KUKA KRL program: EPS_2_25716_MHDR04_A_20250926070356.src

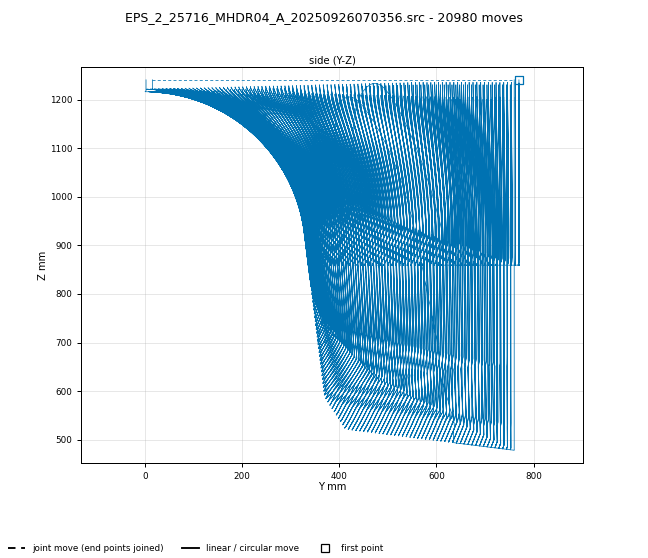
[picture p0: tool path of EPS_2_25716_MHDR04_A_20250926070356.src, 20980 of 20982 moves have a stored position in this frame; points joined in program order, loops and branches not executed]
&ACCESS RVP
&REL 4
&COMMENT QRS 19112012
&PARAM EDITMASK = *
DEF PART()
EXT BAS (BAS_COMMAND :IN,REAL :IN )
INT I
BAS (#INITMOV,0 )

;KUKA QRS Post kuka4.cps  Date:22-06-2017 !

File_ID=2853

QRS_PRE_INIT()

;Init var - Until changes are made in qrs_pre_init
Outlet_Square_prg=0
Inlet_1_Square_prg=0
Inlet_2_Square_prg=0
Inlet_3_Square_prg=0
Inlet_4_Square_prg=0
Inlet_5_Square_prg=0

Outlet_1={X 0.000, Y 562.000, Z 887.500, B 0.000, E1 0.000 }
Inlet_1={X 0.000, Y 612.000, Z 934.000, B 0.000, E1 180.000 }
Outlet_1_type=686
Inlet_1_type=533
;QRS#1=Sidecore dimensions
;QRS#2=675-27" Concrete
;QRS#3=525-21" Concrete
;QRS#4=
;QRS#5=
;QRS#6=
;QRS#7=
;QRS#8=
;QRS#9=S306-38L
;QRS#10=S306-32
;QRS#11=
;QRS#12=
;QRS#13=
;QRS#14=
;QRS#15=
;QRS#16=1524x152x1676 5,5'
;QRS#17=EPS Height
;QRS#18=1230,5
;QRS#19=*
;QRS#20= UPDATED VERSION 22-06-2017
;QRS#21=*
Outlet_Square=0550
Inlet_1_Square=0350
Inlet_2_Square=0
Inlet_3_Square=0
Inlet_4_Square=0
Inlet_5_Square=0
Mill_Square=1
Outlet_Square_Prg=265
Inlet_1_Square_prg=263

QRS_INIT()

$ADVANCE=5

; T1
PTP {E1 171.906,E2 171.906}
PTP {X 0,Y 769.671,A -85,B 0,C 180,E1 171.906,E2 171.906,E3 0,E4 0,E5 0,E6 0}
QRS_SPEED_INIT()
LIN {X 0,Y 769.671,Z 1240.5,A -85,B 0,C 180,E1 171.906,E2 171.906,E3 0,E4 0,E5 0,E6 0} C_VEL
LIN {X 0,Y 769.671,Z 861.31,A -85,B 0,C 180,E1 171.906,E2 171.906} C_VEL
LIN {X 0,Y 769.682,Z 859.31,A -85,B 0,C 180,E1 172.055,E2 172.055} C_VEL
LIN {X 0,Y 770.051,Z 859.31,A -85,B 0,C 180,E1 173.477,E2 173.477} C_VEL
LIN {X 0,Y 770.066,Z 859.31,A -85,B 0,C 180,E1 177.209,E2 177.209} C_VEL
LIN {X 0,Y 770.077,Z 859.31,A -85,B 0,C 180,E1 180.93,E2 180.93} C_VEL
LIN {X 0,Y 770.044,Z 859.31,A -85,B 0,C 180,E1 184.654,E2 184.654} C_VEL
LIN {X 0,Y 770.001,Z 859.31,A -85,B 0,C 180,E1 188.399,E2 188.399} C_VEL
LIN {X 0,Y 769.978,Z 859.31,A -85,B 0,C 180,E1 192.181,E2 192.181} C_VEL
LIN {X 0,Y 769.977,Z 859.31,A -85,B 0,C 180,E1 196.017,E2 196.017} C_VEL
LIN {X 0,Y 769.85,Z 859.31,A -85,B 0,C 180,E1 196.72,E2 196.72} C_VEL
LIN {X 0,Y 769.988,Z 859.31,A -85,B 0,C 180,E1 199.928,E2 199.928} C_VEL
LIN {X 0,Y 769.595,Z 859.31,A -85,B 0,C 180,E1 202.247,E2 202.247} C_VEL
LIN {X 0,Y 769.967,Z 859.31,A -85,B 0,C 180,E1 203.939,E2 203.939} C_VEL
LIN {X 0,Y 769.591,Z 859.31,A -85,B 0,C 180,E1 206.736,E2 206.736} C_VEL
LIN {X 0,Y 769.937,Z 859.31,A -85,B 0,C 180,E1 208.08,E2 208.08} C_VEL
LIN {X 0,Y 769.495,Z 859.31,A -85,B 0,C 180,E1 210.602,E2 210.602} C_VEL
LIN {X 0,Y 769.877,Z 859.31,A -85,B 0,C 180,E1 212.39,E2 212.39} C_VEL
LIN {X 0,Y 769.44,Z 859.31,A -85,B 0,C 180,E1 214.643,E2 214.643} C_VEL
LIN {X 0,Y 770.006,Z 859.31,A -85,B 0,C 180,E1 217.323,E2 217.323} C_VEL
LIN {X 0,Y 769.695,Z 859.31,A -85,B 0,C 180,E1 221.735,E2 221.735} C_VEL
LIN {X 0,Y 769.74,Z 859.31,A -85,B 0,C 180,E1 223.066,E2 223.066} C_VEL
LIN {X 0,Y 769.705,Z 859.31,A -85,B 0,C 180,E1 226.939,E2 226.939} C_VEL
LIN {X 0,Y 769.666,Z 859.31,A -85,B 0,C 180,E1 228.264,E2 228.264} C_VEL
LIN {X 0,Y 770.07,Z 859.31,A -85,B 0,C 180,E1 232.674,E2 232.674} C_VEL
LIN {X 0,Y 769.756,Z 859.31,A -85,B 0,C 180,E1 235.893,E2 235.893} C_VEL
LIN {X 0,Y 769.798,Z 859.31,A -85,B 0,C 180,E1 237.608,E2 237.608} C_VEL
LIN {X 0,Y 770.017,Z 859.31,A -85,B 0,C 180,E1 240.258,E2 240.258} C_VEL
LIN {X 0,Y 769.761,Z 859.31,A -85,B 0,C 180,E1 240.478,E2 240.478} C_VEL
LIN {X 0,Y 767.984,Z 859.31,A -85,B 0,C 180,E1 240.653,E2 240.653} C_VEL
LIN {X 0,Y 768.026,Z 859.947,A -85,B 0,C 180,E1 240.678,E2 240.678} C_VEL
LIN {X 0,Y 769.267,Z 864.427,A -85,B 0,C 180,E1 240.777,E2 240.777} C_VEL
LIN {X 0,Y 769.568,Z 866.732,A -85,B 0,C 180,E1 240.814,E2 240.814} C_VEL
LIN {X 0,Y 769.716,Z 904.713,A -85,B 0,C 180,E1 241.217,E2 241.217} C_VEL
LIN {X 0,Y 769.839,Z 924.965,A -85,B 0,C 180,E1 241.466,E2 241.466} C_VEL
LIN {X 0,Y 769.627,Z 943.026,A -85,B 0,C 180,E1 241.759,E2 241.759} C_VEL
LIN {X 0,Y 769.796,Z 960.577,A -85,B 0,C 180,E1 242.132,E2 242.132} C_VEL
LIN {X 0,Y 769.69,Z 975.698,A -85,B 0,C 180,E1 242.501,E2 242.501} C_VEL
LIN {X 0,Y 769.872,Z 993.181,A -85,B 0,C 180,E1 243.017,E2 243.017} C_VEL
LIN {X 0,Y 769.856,Z 1009.123,A -85,B 0,C 180,E1 243.548,E2 243.548} C_VEL
LIN {X 0,Y 769.815,Z 1019.932,A -85,B 0,C 180,E1 243.947,E2 243.947} C_VEL
LIN {X 0,Y 769.91,Z 1034.617,A -85,B 0,C 180,E1 244.55,E2 244.55} C_VEL
LIN {X 0,Y 769.91,Z 1042.438,A -85,B 0,C 180,E1 244.896,E2 244.896} C_VEL
LIN {X 0,Y 769.862,Z 1054.848,A -85,B 0,C 180,E1 245.478,E2 245.478} C_VEL
LIN {X 0,Y 769.906,Z 1068.593,A -85,B 0,C 180,E1 246.187,E2 246.187} C_VEL
LIN {X 0,Y 769.93,Z 1082.086,A -85,B 0,C 180,E1 246.948,E2 246.948} C_VEL
LIN {X 0,Y 769.915,Z 1094.982,A -85,B 0,C 180,E1 247.739,E2 247.739} C_VEL
LIN {X 0,Y 769.892,Z 1107.85,A -85,B 0,C 180,E1 248.6,E2 248.6} C_VEL
LIN {X 0,Y 769.939,Z 1119.711,A -85,B 0,C 180,E1 249.464,E2 249.464} C_VEL
LIN {X 0,Y 769.935,Z 1130.574,A -85,B 0,C 180,E1 250.319,E2 250.319} C_VEL
LIN {X 0,Y 769.888,Z 1142.058,A -85,B 0,C 180,E1 251.302,E2 251.302} C_VEL
LIN {X 0,Y 769.98,Z 1153.138,A -85,B 0,C 180,E1 252.343,E2 252.343} C_VEL
LIN {X 0,Y 769.834,Z 1162.511,A -85,B 0,C 180,E1 253.29,E2 253.29} C_VEL
LIN {X 0,Y 769.848,Z 1172.264,A -85,B 0,C 180,E1 254.376,E2 254.376} C_VEL
LIN {X 0,Y 769.964,Z 1181.174,A -85,B 0,C 180,E1 255.469,E2 255.469} C_VEL
LIN {X 0,Y 769.771,Z 1189.787,A -85,B 0,C 180,E1 256.624,E2 256.624} C_VEL
LIN {X 0,Y 769.791,Z 1196.239,A -85,B 0,C 180,E1 257.579,E2 257.579} C_VEL
LIN {X 0,Y 769.97,Z 1203.41,A -85,B 0,C 180,E1 258.769,E2 258.769} C_VEL
LIN {X 0,Y 769.805,Z 1209.797,A -85,B 0,C 180,E1 259.95,E2 259.95} C_VEL
LIN {X 0,Y 769.942,Z 1216.32,A -85,B 0,C 180,E1 261.365,E2 261.365} C_VEL
LIN {X 0,Y 769.923,Z 1219.537,A -85,B 0,C 180,E1 262.168,E2 262.168} C_VEL
LIN {X 0,Y 769.786,Z 1222.09,A -85,B 0,C 180,E1 262.857,E2 262.857} C_VEL
LIN {X 0,Y 769.781,Z 1225.359,A -85,B 0,C 180,E1 263.849,E2 263.849} C_VEL
LIN {X 0,Y 769.875,Z 1227.368,A -85,B 0,C 180,E1 264.598,E2 264.598} C_VEL
LIN {X 0,Y 769.915,Z 1229.173,A -85,B 0,C 180,E1 265.345,E2 265.345} C_VEL
LIN {X 0,Y 769.759,Z 1230.789,A -85,B 0,C 180,E1 266.09,E2 266.09} C_VEL
LIN {X 0,Y 769.725,Z 1232.561,A -85,B 0,C 180,E1 267.208,E2 267.208} C_VEL
LIN {X 0,Y 769.922,Z 1233.68,A -85,B 0,C 180,E1 268.326,E2 268.326} C_VEL
LIN {X 0,Y 769.882,Z 1234.171,A -85,B 0,C 180,E1 269.07,E2 269.07} C_VEL
LIN {X 0,Y 769.752,Z 1234.206,A -85,B 0,C 180,E1 270.93,E2 270.93} C_VEL
LIN {X 0,Y 769.983,Z 1233.333,A -85,B 0,C 180,E1 272.046,E2 272.046} C_VEL
LIN {X 0,Y 769.853,Z 1232.527,A -85,B 0,C 180,E1 272.791,E2 272.791} C_VEL
LIN {X 0,Y 769.748,Z 1230.792,A -85,B 0,C 180,E1 273.91,E2 273.91} C_VEL
LIN {X 0,Y 769.834,Z 1229.195,A -85,B 0,C 180,E1 274.656,E2 274.656} C_VEL
LIN {X 0,Y 769.978,Z 1227.341,A -85,B 0,C 180,E1 275.401,E2 275.401} C_VEL
LIN {X 0,Y 769.82,Z 1225.349,A -85,B 0,C 180,E1 276.15,E2 276.15} C_VEL
LIN {X 0,Y 769.746,Z 1221.269,A -85,B 0,C 180,E1 277.393,E2 277.393} C_VEL
LIN {X 0,Y 769.943,Z 1215.307,A -85,B 0,C 180,E1 278.87,E2 278.87} C_VEL
LIN {X 0,Y 769.789,Z 1209.8,A -85,B 0,C 180,E1 280.05,E2 280.05} C_VEL
LIN {X 0,Y 769.876,Z 1203.431,A -85,B 0,C 180,E1 281.232,E2 281.232} C_VEL
LIN {X 0,Y 769.918,Z 1197.677,A -85,B 0,C 180,E1 282.181,E2 282.181} C_VEL
LIN {X 0,Y 769.805,Z 1193.003,A -85,B 0,C 180,E1 282.898,E2 282.898} C_VEL
LIN {X 0,Y 769.803,Z 1188.107,A -85,B 0,C 180,E1 283.614,E2 283.614} C_VEL
LIN {X 0,Y 769.984,Z 1178.906,A -85,B 0,C 180,E1 284.816,E2 284.816} C_VEL
LIN {X 0,Y 769.839,Z 1170.607,A -85,B 0,C 180,E1 285.819,E2 285.819} C_VEL
LIN {X 0,Y 769.821,Z 1160.767,A -85,B 0,C 180,E1 286.894,E2 286.894} C_VEL
LIN {X 0,Y 769.967,Z 1150.001,A -85,B 0,C 180,E1 287.961,E2 287.961} C_VEL
LIN {X 0,Y 769.878,Z 1139.267,A -85,B 0,C 180,E1 288.944,E2 288.944} C_VEL
LIN {X 0,Y 769.906,Z 1129.048,A -85,B 0,C 180,E1 289.806,E2 289.806} C_VEL
LIN {X 0,Y 769.942,Z 1116.517,A -85,B 0,C 180,E1 290.773,E2 290.773} C_VEL
LIN {X 0,Y 769.9,Z 1105.284,A -85,B 0,C 180,E1 291.577,E2 291.577} C_VEL
LIN {X 0,Y 769.914,Z 1092.612,A -85,B 0,C 180,E1 292.411,E2 292.411} C_VEL
LIN {X 0,Y 769.921,Z 1078.814,A -85,B 0,C 180,E1 293.242,E2 293.242} C_VEL
LIN {X 0,Y 769.909,Z 1064.631,A -85,B 0,C 180,E1 294.023,E2 294.023} C_VEL
LIN {X 0,Y 769.846,Z 1051.463,A -85,B 0,C 180,E1 294.69,E2 294.69} C_VEL
LIN {X 0,Y 769.909,Z 1036.961,A -85,B 0,C 180,E1 295.353,E2 295.353} C_VEL
LIN {X 0,Y 769.869,Z 1020.065,A -85,B 0,C 180,E1 296.046,E2 296.046} C_VEL
LIN {X 0,Y 769.811,Z 1007.364,A -85,B 0,C 180,E1 296.519,E2 296.519} C_VEL
LIN {X 0,Y 769.897,Z 989.325,A -85,B 0,C 180,E1 297.102,E2 297.102} C_VEL
LIN {X 0,Y 769.783,Z 972.607,A -85,B 0,C 180,E1 297.575,E2 297.575} C_VEL
LIN {X 0,Y 769.703,Z 963.365,A -85,B 0,C 180,E1 297.804,E2 297.804} C_VEL
LIN {X 0,Y 769.829,Z 954.273,A -85,B 0,C 180,E1 298.005,E2 298.005} C_VEL
LIN {X 0,Y 769.853,Z 939.702,A -85,B 0,C 180,E1 298.293,E2 298.293} C_VEL
LIN {X 0,Y 769.612,Z 922.786,A -85,B 0,C 180,E1 298.571,E2 298.571} C_VEL
LIN {X 0,Y 769.691,Z 903.386,A -85,B 0,C 180,E1 298.798,E2 298.798} C_VEL
LIN {X 0,Y 769.594,Z 868.345,A -85,B 0,C 180,E1 299.168,E2 299.168} C_VEL
LIN {X 0,Y 769.47,Z 865.258,A -85,B 0,C 180,E1 299.206,E2 299.206} C_VEL
LIN {X 0,Y 768.381,Z 860.967,A -85,B 0,C 180,E1 299.296,E2 299.296} C_VEL
LIN {X 0,Y 767.894,Z 859.31,A -85,B 0,C 180,E1 299.344,E2 299.344} C_VEL
LIN {X 0,Y 768.202,Z 859.31,A -85,B 0,C 180,E1 299.358,E2 299.358} C_VEL
LIN {X 0,Y 769.579,Z 859.31,A -85,B 0,C 180,E1 299.487,E2 299.487} C_VEL
LIN {X 0,Y 770.036,Z 859.31,A -85,B 0,C 180,E1 299.696,E2 299.696} C_VEL
LIN {X 0,Y 769.962,Z 859.31,A -85,B 0,C 180,E1 302.384,E2 302.384} C_VEL
LIN {X 0,Y 769.489,Z 859.31,A -85,B 0,C 180,E1 304.639,E2 304.639} C_VEL
LIN {X 0,Y 770.073,Z 859.31,A -85,B 0,C 180,E1 307.326,E2 307.326} C_VEL
LIN {X 0,Y 769.766,Z 859.31,A -85,B 0,C 180,E1 311.729,E2 311.729} C_VEL
LIN {X 0,Y 769.826,Z 859.31,A -85,B 0,C 180,E1 313.071,E2 313.071} C_VEL
LIN {X 0,Y 769.84,Z 859.31,A -85,B 0,C 180,E1 314.267,E2 314.267} C_VEL
LIN {X 0,Y 769.763,Z 859.31,A -85,B 0,C 180,E1 315.725,E2 315.725} C_VEL
LIN {X 0,Y 769.763,Z 859.31,A -85,B 0,C 180,E1 319.731,E2 319.731} C_VEL
LIN {X 0,Y 769.807,Z 859.31,A -85,B 0,C 180,E1 320.719,E2 320.719} C_VEL
LIN {X 0,Y 769.409,Z 859.31,A -85,B 0,C 180,E1 323.061,E2 323.061} C_VEL
LIN {X 0,Y 769.837,Z 859.31,A -85,B 0,C 180,E1 325.377,E2 325.377} C_VEL
LIN {X 0,Y 770.001,Z 859.31,A -85,B 0,C 180,E1 329.334,E2 329.334} C_VEL
LIN {X 0,Y 769.842,Z 859.31,A -85,B 0,C 180,E1 333.227,E2 333.227} C_VEL
LIN {X 0,Y 769.935,Z 859.31,A -85,B 0,C 180,E1 334.008,E2 334.008} C_VEL
LIN {X 0,Y 769.999,Z 859.31,A -85,B 0,C 180,E1 337.68,E2 337.68} C_VEL
LIN {X 0,Y 769.97,Z 859.31,A -85,B 0,C 180,E1 338.08,E2 338.08} C_VEL
LIN {X 0,Y 769.98,Z 859.31,A -85,B 0,C 180,E1 342.039,E2 342.039} C_VEL
LIN {X 0,Y 769.696,Z 859.31,A -85,B 0,C 180,E1 343.977,E2 343.977} C_VEL
LIN {X 0,Y 769.78,Z 859.31,A -85,B 0,C 180,E1 345.906,E2 345.906} C_VEL
LIN {X 0,Y 769.98,Z 859.31,A -85,B 0,C 180,E1 349.716,E2 349.716} C_VEL
LIN {X 0,Y 770.006,Z 859.31,A -85,B 0,C 180,E1 353.477,E2 353.477} C_VEL
LIN {X 0,Y 770.059,Z 859.31,A -85,B 0,C 180,E1 357.209,E2 357.209} C_VEL
LIN {X 0,Y 770.073,Z 859.31,A -85,B 0,C 180,E1 360.93,E2 360.93} C_VEL
LIN {X 0,Y 770.057,Z 859.31,A -85,B 0,C 180,E1 364.654,E2 364.654} C_VEL
LIN {X 0,Y 770.018,Z 859.31,A -85,B 0,C 180,E1 368.399,E2 368.399} C_VEL
LIN {X 0,Y 769.982,Z 859.31,A -85,B 0,C 180,E1 372.181,E2 372.181} C_VEL
LIN {X 0,Y 769.963,Z 859.31,A -85,B 0,C 180,E1 376.017,E2 376.017} C_VEL
LIN {X 0,Y 769.829,Z 859.31,A -85,B 0,C 180,E1 376.715,E2 376.715} C_VEL
LIN {X 0,Y 769.937,Z 859.31,A -85,B 0,C 180,E1 379.929,E2 379.929} C_VEL
LIN {X 0,Y 769.562,Z 859.31,A -85,B 0,C 180,E1 382.241,E2 382.241} C_VEL
LIN {X 0,Y 769.917,Z 859.31,A -85,B 0,C 180,E1 383.941,E2 383.941} C_VEL
LIN {X 0,Y 769.542,Z 859.31,A -85,B 0,C 180,E1 386.729,E2 386.729} C_VEL
LIN {X 0,Y 769.888,Z 859.31,A -85,B 0,C 180,E1 388.082,E2 388.082} C_VEL
LIN {X 0,Y 769.488,Z 859.31,A -85,B 0,C 180,E1 390.601,E2 390.601} C_VEL
LIN {X 0,Y 769.865,Z 859.31,A -85,B 0,C 180,E1 392.39,E2 392.39} C_VEL
LIN {X 0,Y 769.445,Z 859.31,A -85,B 0,C 180,E1 394.643,E2 394.643} C_VEL
LIN {X 0,Y 770.04,Z 859.31,A -85,B 0,C 180,E1 397.326,E2 397.326} C_VEL
LIN {X 0,Y 769.705,Z 859.31,A -85,B 0,C 180,E1 401.735,E2 401.735} C_VEL
LIN {X 0,Y 769.752,Z 859.31,A -85,B 0,C 180,E1 403.067,E2 403.067} C_VEL
LIN {X 0,Y 769.737,Z 859.31,A -85,B 0,C 180,E1 406.937,E2 406.937} C_VEL
LIN {X 0,Y 769.692,Z 859.31,A -85,B 0,C 180,E1 408.266,E2 408.266} C_VEL
LIN {X 0,Y 770.062,Z 859.31,A -85,B 0,C 180,E1 412.675,E2 412.675} C_VEL
LIN {X 0,Y 769.748,Z 859.31,A -85,B 0,C 180,E1 415.894,E2 415.894} C_VEL
LIN {X 0,Y 769.672,Z 859.31,A -85,B 0,C 180,E1 417.602,E2 417.602} C_VEL
LIN {X 0,Y 769.433,Z 859.31,A -85,B 0,C 180,E1 419.769,E2 419.769} C_VEL
LIN {X 0,Y 769.91,Z 859.31,A -85,B 0,C 180,E1 421.92,E2 421.92} C_VEL
LIN {X 0,Y 770.081,Z 859.31,A -85,B 0,C 180,E1 426.297,E2 426.297} C_VEL
LIN {X 0,Y 769.403,Z 859.31,A -85,B 0,C 180,E1 426.506,E2 426.506} C_VEL
LIN {X 0,Y 768.639,Z 859.31,A -85,B 0,C 180,E1 426.577,E2 426.577} C_VEL
LIN {X 0,Y 769.411,Z 862.963,A -85,B 0,C 180,E1 426.652,E2 426.652} C_VEL
LIN {X 0,Y 769.765,Z 870.896,A -85,B 0,C 180,E1 426.742,E2 426.742} C_VEL
LIN {X 0,Y 769.853,Z 946.408,A -85,B 0,C 180,E1 427.495,E2 427.495} C_VEL
LIN {X 0,Y 769.952,Z 960.871,A -85,B 0,C 180,E1 427.677,E2 427.677} C_VEL
LIN {X 0,Y 769.864,Z 974.295,A -85,B 0,C 180,E1 427.892,E2 427.892} C_VEL
LIN {X 0,Y 769.934,Z 984.387,A -85,B 0,C 180,E1 428.089,E2 428.089} C_VEL
LIN {X 0,Y 769.985,Z 999.962,A -85,B 0,C 180,E1 428.458,E2 428.458} C_VEL
LIN {X 0,Y 769.905,Z 1013.381,A -85,B 0,C 180,E1 428.83,E2 428.83} C_VEL
LIN {X 0,Y 769.957,Z 1025.148,A -85,B 0,C 180,E1 429.206,E2 429.206} C_VEL
LIN {X 0,Y 769.979,Z 1038.217,A -85,B 0,C 180,E1 429.68,E2 429.68} C_VEL
LIN {X 0,Y 769.926,Z 1049.488,A -85,B 0,C 180,E1 430.133,E2 430.133} C_VEL
LIN {X 0,Y 769.981,Z 1061.815,A -85,B 0,C 180,E1 430.69,E2 430.69} C_VEL
LIN {X 0,Y 769.982,Z 1072.942,A -85,B 0,C 180,E1 431.243,E2 431.243} C_VEL
LIN {X 0,Y 769.967,Z 1084.12,A -85,B 0,C 180,E1 431.855,E2 431.855} C_VEL
LIN {X 0,Y 769.957,Z 1094.576,A -85,B 0,C 180,E1 432.483,E2 432.483} C_VEL
LIN {X 0,Y 769.955,Z 1104.699,A -85,B 0,C 180,E1 433.149,E2 433.149} C_VEL
LIN {X 0,Y 769.998,Z 1113.725,A -85,B 0,C 180,E1 433.794,E2 433.794} C_VEL
LIN {X 0,Y 769.959,Z 1123.75,A -85,B 0,C 180,E1 434.577,E2 434.577} C_VEL
LIN {X 0,Y 769.898,Z 1131.942,A -85,B 0,C 180,E1 435.272,E2 435.272} C_VEL
LIN {X 0,Y 769.96,Z 1140.118,A -85,B 0,C 180,E1 436.029,E2 436.029} C_VEL
LIN {X 0,Y 769.949,Z 1148.387,A -85,B 0,C 180,E1 436.866,E2 436.866} C_VEL
LIN {X 0,Y 769.87,Z 1155.915,A -85,B 0,C 180,E1 437.699,E2 437.699} C_VEL
LIN {X 0,Y 769.914,Z 1162.733,A -85,B 0,C 180,E1 438.531,E2 438.531} C_VEL
LIN {X 0,Y 769.978,Z 1168.094,A -85,B 0,C 180,E1 439.243,E2 439.243} C_VEL
LIN {X 0,Y 769.844,Z 1174.555,A -85,B 0,C 180,E1 440.186,E2 440.186} C_VEL
LIN {X 0,Y 769.866,Z 1180.255,A -85,B 0,C 180,E1 441.129,E2 441.129} C_VEL
LIN {X 0,Y 769.951,Z 1185.836,A -85,B 0,C 180,E1 442.192,E2 442.192} C_VEL
LIN {X 0,Y 769.81,Z 1190.358,A -85,B 0,C 180,E1 443.172,E2 443.172} C_VEL
LIN {X 0,Y 769.845,Z 1194.421,A -85,B 0,C 180,E1 444.224,E2 444.224} C_VEL
LIN {X 0,Y 769.974,Z 1196.895,A -85,B 0,C 180,E1 444.972,E2 444.972} C_VEL
LIN {X 0,Y 769.82,Z 1199.939,A -85,B 0,C 180,E1 446.091,E2 446.091} C_VEL
LIN {X 0,Y 769.843,Z 1202.142,A -85,B 0,C 180,E1 447.209,E2 447.209} C_VEL
LIN {X 0,Y 769.986,Z 1203.212,A -85,B 0,C 180,E1 447.954,E2 447.954} C_VEL
LIN {X 0,Y 769.799,Z 1204.215,A -85,B 0,C 180,E1 449.07,E2 449.07} C_VEL
LIN {X 0,Y 769.84,Z 1204.172,A -85,B 0,C 180,E1 450.93,E2 450.93} C_VEL
LIN {X 0,Y 769.988,Z 1203.478,A -85,B 0,C 180,E1 451.674,E2 451.674} C_VEL
LIN {X 0,Y 769.807,Z 1202.02,A -85,B 0,C 180,E1 452.791,E2 452.791} C_VEL
LIN {X 0,Y 769.853,Z 1199.737,A -85,B 0,C 180,E1 453.909,E2 453.909} C_VEL
LIN {X 0,Y 769.949,Z 1196.599,A -85,B 0,C 180,E1 455.028,E2 455.028} C_VEL
LIN {X 0,Y 769.846,Z 1194.12,A -85,B 0,C 180,E1 455.776,E2 455.776} C_VEL
LIN {X 0,Y 769.885,Z 1190.021,A -85,B 0,C 180,E1 456.818,E2 456.818} C_VEL
LIN {X 0,Y 769.948,Z 1185.617,A -85,B 0,C 180,E1 457.765,E2 457.765} C_VEL
LIN {X 0,Y 769.837,Z 1179.731,A -85,B 0,C 180,E1 458.871,E2 458.871} C_VEL
LIN {X 0,Y 769.928,Z 1173.935,A -85,B 0,C 180,E1 459.812,E2 459.812} C_VEL
LIN {X 0,Y 769.961,Z 1167.417,A -85,B 0,C 180,E1 460.757,E2 460.757} C_VEL
LIN {X 0,Y 769.874,Z 1160.128,A -85,B 0,C 180,E1 461.707,E2 461.707} C_VEL
LIN {X 0,Y 769.934,Z 1153.042,A -85,B 0,C 180,E1 462.538,E2 462.538} C_VEL
LIN {X 0,Y 769.957,Z 1145.234,A -85,B 0,C 180,E1 463.373,E2 463.373} C_VEL
LIN {X 0,Y 769.901,Z 1137.956,A -85,B 0,C 180,E1 464.092,E2 464.092} C_VEL
LIN {X 0,Y 769.937,Z 1128.885,A -85,B 0,C 180,E1 464.905,E2 464.905} C_VEL
LIN {X 0,Y 769.974,Z 1120.313,A -85,B 0,C 180,E1 465.611,E2 465.611} C_VEL
LIN {X 0,Y 769.955,Z 1111.181,A -85,B 0,C 180,E1 466.304,E2 466.304} C_VEL
LIN {X 0,Y 769.981,Z 1101.105,A -85,B 0,C 180,E1 467.003,E2 467.003} C_VEL
LIN {X 0,Y 769.987,Z 1090.68,A -85,B 0,C 180,E1 467.665,E2 467.665} C_VEL
LIN {X 0,Y 769.967,Z 1080.354,A -85,B 0,C 180,E1 468.267,E2 468.267} C_VEL
LIN {X 0,Y 769.962,Z 1070.009,A -85,B 0,C 180,E1 468.819,E2 468.819} C_VEL
LIN {X 0,Y 769.921,Z 1058.587,A -85,B 0,C 180,E1 469.373,E2 469.373} C_VEL
LIN {X 0,Y 769.976,Z 1045.821,A -85,B 0,C 180,E1 469.927,E2 469.927} C_VEL
LIN {X 0,Y 769.957,Z 1033.547,A -85,B 0,C 180,E1 470.406,E2 470.406} C_VEL
LIN {X 0,Y 769.893,Z 1021.715,A -85,B 0,C 180,E1 470.82,E2 470.82} C_VEL
LIN {X 0,Y 769.973,Z 1009.361,A -85,B 0,C 180,E1 471.197,E2 471.197} C_VEL
LIN {X 0,Y 769.926,Z 995.328,A -85,B 0,C 180,E1 471.569,E2 471.569} C_VEL
LIN {X 0,Y 769.895,Z 984.757,A -85,B 0,C 180,E1 471.815,E2 471.815} C_VEL
LIN {X 0,Y 769.941,Z 969.253,A -85,B 0,C 180,E1 472.103,E2 472.103} C_VEL
LIN {X 0,Y 769.8,Z 956.534,A -85,B 0,C 180,E1 472.298,E2 472.298} C_VEL
LIN {X 0,Y 769.828,Z 938.257,A -85,B 0,C 180,E1 472.498,E2 472.498} C_VEL
LIN {X 0,Y 769.621,Z 860.007,A -85,B 0,C 180,E1 473.281,E2 473.281} C_VEL
LIN {X 0,Y 769.775,Z 859.31,A -85,B 0,C 180,E1 473.311,E2 473.311} C_VEL
LIN {X 0,Y 770.073,Z 859.31,A -85,B 0,C 180,E1 473.407,E2 473.407} C_VEL
LIN {X 0,Y 769.916,Z 859.31,A -85,B 0,C 180,E1 478.08,E2 478.08} C_VEL
LIN {X 0,Y 769.504,Z 859.31,A -85,B 0,C 180,E1 480.6,E2 480.6} C_VEL
LIN {X 0,Y 769.877,Z 859.31,A -85,B 0,C 180,E1 482.388,E2 482.388} C_VEL
LIN {X 0,Y 769.547,Z 859.31,A -85,B 0,C 180,E1 484.084,E2 484.084} C_VEL
LIN {X 0,Y 770.042,Z 859.31,A -85,B 0,C 180,E1 487.324,E2 487.324} C_VEL
LIN {X 0,Y 769.814,Z 859.31,A -85,B 0,C 180,E1 491.726,E2 491.726} C_VEL
LIN {X 0,Y 769.657,Z 859.31,A -85,B 0,C 180,E1 493.057,E2 493.057} C_VEL
LIN {X 0,Y 769.736,Z 859.31,A -85,B 0,C 180,E1 496.934,E2 496.934} C_VEL
LIN {X 0,Y 769.706,Z 859.31,A -85,B 0,C 180,E1 498.265,E2 498.265} C_VEL
LIN {X 0,Y 770.043,Z 859.31,A -85,B 0,C 180,E1 502.674,E2 502.674} C_VEL
LIN {X 0,Y 769.741,Z 859.31,A -85,B 0,C 180,E1 505.892,E2 505.892} C_VEL
LIN {X 0,Y 769.67,Z 859.31,A -85,B 0,C 180,E1 507.601,E2 507.601} C_VEL
LIN {X 0,Y 769.411,Z 859.31,A -85,B 0,C 180,E1 509.767,E2 509.767} C_VEL
LIN {X 0,Y 769.917,Z 859.31,A -85,B 0,C 180,E1 511.919,E2 511.919} C_VEL
LIN {X 0,Y 769.558,Z 859.31,A -85,B 0,C 180,E1 513.994,E2 513.994} C_VEL
LIN {X 0,Y 769.947,Z 859.31,A -85,B 0,C 180,E1 516.06,E2 516.06} C_VEL
LIN {X 0,Y 769.576,Z 859.31,A -85,B 0,C 180,E1 518.069,E2 518.069} C_VEL
LIN {X 0,Y 769.928,Z 859.31,A -85,B 0,C 180,E1 520.071,E2 520.071} C_VEL
LIN {X 0,Y 769.407,Z 859.31,A -85,B 0,C 180,E1 523.971,E2 523.971} C_VEL
LIN {X 0,Y 769.813,Z 859.31,A -85,B 0,C 180,E1 525.906,E2 525.906} C_VEL
LIN {X 0,Y 770.001,Z 859.31,A -85,B 0,C 180,E1 529.716,E2 529.716} C_VEL
LIN {X 0,Y 769.682,Z 859.31,A -85,B 0,C 180,E1 532.055,E2 532.055} C_VEL
LIN {X 0,Y 765.849,Z 859.31,A -85,B 0,C 180,E1 533.331,E2 533.331} C_VEL
LIN {X 0,Y 761.824,Z 859.31,A -85,B 0,C 180,E1 534.62,E2 534.62} C_VEL
LIN {X 0,Y 761.801,Z 859.31,A -85,B 0,C 180,E1 538.862,E2 538.862} C_VEL
LIN {X 0,Y 761.796,Z 859.31,A -85,B 0,C 180,E1 542.281,E2 542.281} C_VEL
LIN {X 0,Y 761.785,Z 859.31,A -85,B 0,C 180,E1 545.973,E2 545.973} C_VEL
LIN {X 0,Y 761.68,Z 859.31,A -85,B 0,C 180,E1 550.313,E2 550.313} C_VEL
LIN {X 0,Y 761.657,Z 859.31,A -85,B 0,C 180,E1 553.81,E2 553.81} C_VEL
LIN {X 0,Y 761.803,Z 859.31,A -85,B 0,C 180,E1 557.356,E2 557.356} C_VEL
LIN {X 0,Y 761.779,Z 859.31,A -85,B 0,C 180,E1 560.976,E2 560.976} C_VEL
LIN {X 0,Y 761.795,Z 859.31,A -85,B 0,C 180,E1 564.685,E2 564.685} C_VEL
LIN {X 0,Y 761.74,Z 859.31,A -85,B 0,C 180,E1 568.923,E2 568.923} C_VEL
LIN {X 0,Y 761.661,Z 859.31,A -85,B 0,C 180,E1 573.324,E2 573.324} C_VEL
LIN {X 0,Y 761.738,Z 859.31,A -85,B 0,C 180,E1 578.063,E2 578.063} C_VEL
LIN {X 0,Y 761.808,Z 859.31,A -85,B 0,C 180,E1 582.612,E2 582.612} C_VEL
LIN {X 0,Y 761.763,Z 859.31,A -85,B 0,C 180,E1 587.443,E2 587.443} C_VEL
LIN {X 0,Y 761.924,Z 859.31,A -85,B 0,C 180,E1 593.371,E2 593.371} C_VEL
LIN {X 0,Y 761.887,Z 859.31,A -85,B 0,C 180,E1 597.521,E2 597.521} C_VEL
LIN {X 0,Y 761.341,Z 859.31,A -85,B 0,C 180,E1 600.333,E2 600.333} C_VEL
LIN {X 0,Y 762.681,Z 873.024,A -85,B 0,C 180,E1 600.591,E2 600.591} C_VEL
LIN {X 0,Y 762.731,Z 940.184,A -85,B 0,C 180,E1 601.427,E2 601.427} C_VEL
LIN {X 0,Y 762.679,Z 984.756,A -85,B 0,C 180,E1 602.488,E2 602.488} C_VEL
LIN {X 0,Y 762.618,Z 1026.505,A -85,B 0,C 180,E1 603.948,E2 603.948} C_VEL
LIN {X 0,Y 762.493,Z 1068.015,A -85,B 0,C 180,E1 605.908,E2 605.908} C_VEL
LIN {X 0,Y 762.316,Z 1107.451,A -85,B 0,C 180,E1 608.347,E2 608.347} C_VEL
LIN {X 0,Y 762.188,Z 1142.627,A -85,B 0,C 180,E1 611.152,E2 611.152} C_VEL
LIN {X 0,Y 762.09,Z 1171.881,A -85,B 0,C 180,E1 614.133,E2 614.133} C_VEL
LIN {X 0,Y 761.965,Z 1196.137,A -85,B 0,C 180,E1 617.364,E2 617.364} C_VEL
LIN {X 0,Y 762.01,Z 1212.484,A -85,B 0,C 180,E1 620.269,E2 620.269} C_VEL
LIN {X 0,Y 761.964,Z 1225.197,A -85,B 0,C 180,E1 623.457,E2 623.457} C_VEL
LIN {X 0,Y 761.905,Z 1232.65,A -85,B 0,C 180,E1 626.579,E2 626.579} C_VEL
LIN {X 0,Y 761.945,Z 1235.5,A -85,B 0,C 180,E1 630,E2 630} C_VEL
LIN {X 0,Y 761.954,Z 1232.651,A -85,B 0,C 180,E1 633.42,E2 633.42} C_VEL
LIN {X 0,Y 762.009,Z 1226.123,A -85,B 0,C 180,E1 636.26,E2 636.26} C_VEL
LIN {X 0,Y 762.013,Z 1212.486,A -85,B 0,C 180,E1 639.731,E2 639.731} C_VEL
LIN {X 0,Y 762.019,Z 1194.14,A -85,B 0,C 180,E1 642.931,E2 642.931} C_VEL
LIN {X 0,Y 762.07,Z 1171.884,A -85,B 0,C 180,E1 645.867,E2 645.867} C_VEL
LIN {X 0,Y 762.187,Z 1140.996,A -85,B 0,C 180,E1 648.999,E2 648.999} C_VEL
LIN {X 0,Y 762.345,Z 1106.382,A -85,B 0,C 180,E1 651.728,E2 651.728} C_VEL
LIN {X 0,Y 762.517,Z 1066.311,A -85,B 0,C 180,E1 654.185,E2 654.185} C_VEL
LIN {X 0,Y 762.657,Z 1023.414,A -85,B 0,C 180,E1 656.181,E2 656.181} C_VEL
LIN {X 0,Y 762.747,Z 980.597,A -85,B 0,C 180,E1 657.629,E2 657.629} C_VEL
LIN {X 0,Y 762.866,Z 938.992,A -85,B 0,C 180,E1 658.587,E2 658.587} C_VEL
LIN {X 0,Y 762.72,Z 884.129,A -85,B 0,C 180,E1 659.29,E2 659.29} C_VEL
LIN {X 0,Y 761.984,Z 864.462,A -85,B 0,C 180,E1 659.53,E2 659.53} C_VEL
LIN {X 0,Y 761.014,Z 859.31,A -85,B 0,C 180,E1 659.634,E2 659.634} C_VEL
LIN {X 0,Y 762.115,Z 859.31,A -85,B 0,C 180,E1 659.806,E2 659.806} C_VEL
LIN {X 0,Y 761.642,Z 859.31,A -85,B 0,C 180,E1 663.853,E2 663.853} C_VEL
LIN {X 0,Y 761.799,Z 859.31,A -85,B 0,C 180,E1 668.07,E2 668.07} C_VEL
LIN {X 0,Y 761.86,Z 859.31,A -85,B 0,C 180,E1 672.63,E2 672.63} C_VEL
LIN {X 0,Y 761.796,Z 859.31,A -85,B 0,C 180,E1 675.891,E2 675.891} C_VEL
LIN {X 0,Y 761.856,Z 859.31,A -85,B 0,C 180,E1 680.867,E2 680.867} C_VEL
LIN {X 0,Y 761.68,Z 859.31,A -85,B 0,C 180,E1 686.157,E2 686.157} C_VEL
LIN {X 0,Y 761.781,Z 859.31,A -85,B 0,C 180,E1 690.186,E2 690.186} C_VEL
LIN {X 0,Y 762.01,Z 859.31,A -85,B 0,C 180,E1 694.062,E2 694.062} C_VEL
LIN {X 0,Y 762.116,Z 859.31,A -85,B 0,C 180,E1 697.809,E2 697.809} C_VEL
LIN {X 0,Y 761.906,Z 859.31,A -85,B 0,C 180,E1 702.675,E2 702.675} C_VEL
LIN {X 0,Y 761.556,Z 859.31,A -85,B 0,C 180,E1 707.359,E2 707.359} C_VEL
LIN {X 0,Y 761.749,Z 859.31,A -85,B 0,C 180,E1 710.844,E2 710.844} C_VEL
LIN {X 0,Y 761.838,Z 859.31,A -85,B 0,C 180,E1 714.292,E2 714.292} C_VEL
LIN {X 0,Y 761.768,Z 859.31,A -85,B 0,C 180,E1 718.859,E2 718.859} C_VEL
LIN {X 0,Y 761.803,Z 859.31,A -85,B 0,C 180,E1 722.278,E2 722.278} C_VEL
LIN {X 0,Y 761.793,Z 859.31,A -85,B 0,C 180,E1 725.982,E2 725.982} C_VEL
LIN {X 0,Y 761.706,Z 859.31,A -85,B 0,C 180,E1 730.31,E2 730.31} C_VEL
LIN {X 0,Y 761.664,Z 859.31,A -85,B 0,C 180,E1 733.806,E2 733.806} C_VEL
LIN {X 0,Y 761.779,Z 859.31,A -85,B 0,C 180,E1 737.353,E2 737.353} C_VEL
LIN {X 0,Y 761.716,Z 859.31,A -85,B 0,C 180,E1 740.975,E2 740.975} C_VEL
LIN {X 0,Y 761.747,Z 859.31,A -85,B 0,C 180,E1 744.683,E2 744.683} C_VEL
LIN {X 0,Y 761.714,Z 859.31,A -85,B 0,C 180,E1 748.92,E2 748.92} C_VEL
LIN {X 0,Y 761.651,Z 859.31,A -85,B 0,C 180,E1 753.324,E2 753.324} C_VEL
LIN {X 0,Y 761.773,Z 859.31,A -85,B 0,C 180,E1 758.057,E2 758.057} C_VEL
LIN {X 0,Y 761.791,Z 859.31,A -85,B 0,C 180,E1 762.611,E2 762.611} C_VEL
LIN {X 0,Y 761.772,Z 859.31,A -85,B 0,C 180,E1 767.444,E2 767.444} C_VEL
LIN {X 0,Y 761.904,Z 859.31,A -85,B 0,C 180,E1 773.37,E2 773.37} C_VEL
LIN {X 0,Y 761.789,Z 859.31,A -85,B 0,C 180,E1 777.516,E2 777.516} C_VEL
LIN {X 0,Y 761.7,Z 859.31,A -85,B 0,C 180,E1 782.771,E2 782.771} C_VEL
LIN {X 0,Y 761.376,Z 859.31,A -85,B 0,C 180,E1 786.346,E2 786.346} C_VEL
LIN {X 0,Y 762.531,Z 893.643,A -85,B 0,C 180,E1 786.737,E2 786.737} C_VEL
LIN {X 0,Y 762.593,Z 969.685,A -85,B 0,C 180,E1 787.588,E2 787.588} C_VEL
LIN {X 0,Y 762.546,Z 1010.612,A -85,B 0,C 180,E1 788.53,E2 788.53} C_VEL
LIN {X 0,Y 762.396,Z 1049.948,A -85,B 0,C 180,E1 789.949,E2 789.949} C_VEL
LIN {X 0,Y 762.347,Z 1084.745,A -85,B 0,C 180,E1 791.704,E2 791.704} C_VEL
LIN {X 0,Y 762.292,Z 1116.647,A -85,B 0,C 180,E1 793.842,E2 793.842} C_VEL
LIN {X 0,Y 762.191,Z 1143.565,A -85,B 0,C 180,E1 796.198,E2 796.198} C_VEL
LIN {X 0,Y 762.146,Z 1166.33,A -85,B 0,C 180,E1 798.823,E2 798.823} C_VEL
LIN {X 0,Y 762.07,Z 1184.568,A -85,B 0,C 180,E1 801.712,E2 801.712} C_VEL
LIN {X 0,Y 762.027,Z 1195.752,A -85,B 0,C 180,E1 804.294,E2 804.294} C_VEL
LIN {X 0,Y 761.973,Z 1202.02,A -85,B 0,C 180,E1 806.58,E2 806.58} C_VEL
LIN {X 0,Y 761.988,Z 1205.12,A -85,B 0,C 180,E1 808.861,E2 808.861} C_VEL
LIN {X 0,Y 762.04,Z 1205.041,A -85,B 0,C 180,E1 811.14,E2 811.14} C_VEL
LIN {X 0,Y 762.056,Z 1200.599,A -85,B 0,C 180,E1 813.991,E2 813.991} C_VEL
LIN {X 0,Y 762.075,Z 1189.716,A -85,B 0,C 180,E1 817.139,E2 817.139} C_VEL
LIN {X 0,Y 762.114,Z 1173.852,A -85,B 0,C 180,E1 820.019,E2 820.019} C_VEL
LIN {X 0,Y 762.171,Z 1152.453,A -85,B 0,C 180,E1 822.777,E2 822.777} C_VEL
LIN {X 0,Y 762.215,Z 1126.556,A -85,B 0,C 180,E1 825.273,E2 825.273} C_VEL
LIN {X 0,Y 762.311,Z 1096.643,A -85,B 0,C 180,E1 827.476,E2 827.476} C_VEL
LIN {X 0,Y 762.388,Z 1062.808,A -85,B 0,C 180,E1 829.371,E2 829.371} C_VEL
LIN {X 0,Y 762.485,Z 1025.006,A -85,B 0,C 180,E1 830.922,E2 830.922} C_VEL
LIN {X 0,Y 762.544,Z 985.099,A -85,B 0,C 180,E1 832.029,E2 832.029} C_VEL
LIN {X 0,Y 762.546,Z 946.198,A -85,B 0,C 180,E1 832.645,E2 832.645} C_VEL
LIN {X 0,Y 762.091,Z 859.31,A -85,B 0,C 180,E1 833.542,E2 833.542} C_VEL
LIN {X 0,Y 761.715,Z 859.31,A -85,B 0,C 180,E1 838.95,E2 838.95} C_VEL
LIN {X 0,Y 761.725,Z 859.31,A -85,B 0,C 180,E1 843.358,E2 843.358} C_VEL
LIN {X 0,Y 761.785,Z 859.31,A -85,B 0,C 180,E1 848.071,E2 848.071} C_VEL
LIN {X 0,Y 761.763,Z 859.31,A -85,B 0,C 180,E1 852.627,E2 852.627} C_VEL
LIN {X 0,Y 761.794,Z 859.31,A -85,B 0,C 180,E1 857.461,E2 857.461} C_VEL
LIN {X 0,Y 761.871,Z 859.31,A -85,B 0,C 180,E1 863.381,E2 863.381} C_VEL
LIN {X 0,Y 761.774,Z 859.31,A -85,B 0,C 180,E1 867.527,E2 867.527} C_VEL
LIN {X 0,Y 761.745,Z 859.31,A -85,B 0,C 180,E1 872.782,E2 872.782} C_VEL
LIN {X 0,Y 761.881,Z 859.31,A -85,B 0,C 180,E1 876.569,E2 876.569} C_VEL
LIN {X 0,Y 761.952,Z 859.31,A -85,B 0,C 180,E1 880.247,E2 880.247} C_VEL
LIN {X 0,Y 761.834,Z 859.31,A -85,B 0,C 180,E1 886.197,E2 886.197} C_VEL
LIN {X 0,Y 761.786,Z 859.31,A -85,B 0,C 180,E1 890.848,E2 890.848} C_VEL
LIN {X 0,Y 761.824,Z 859.31,A -85,B 0,C 180,E1 894.62,E2 894.62} C_VEL
LIN {X 0,Y 757.857,Z 859.31,A -85,B 0,C 180,E1 895.903,E2 895.903} C_VEL
LIN {X 0,Y 754.025,Z 859.31,A -85,B 0,C 180,E1 897.199,E2 897.199} C_VEL
LIN {X 0,Y 753.902,Z 859.31,A -85,B 0,C 180,E1 902.305,E2 902.305} C_VEL
LIN {X 0,Y 753.928,Z 859.31,A -85,B 0,C 180,E1 905.768,E2 905.768} C_VEL
LIN {X 0,Y 753.823,Z 859.31,A -85,B 0,C 180,E1 909.945,E2 909.945} C_VEL
LIN {X 0,Y 753.754,Z 859.31,A -85,B 0,C 180,E1 913.958,E2 913.958} C_VEL
LIN {X 0,Y 753.872,Z 859.31,A -85,B 0,C 180,E1 917.545,E2 917.545} C_VEL
LIN {X 0,Y 753.841,Z 859.31,A -85,B 0,C 180,E1 921.208,E2 921.208} C_VEL
LIN {X 0,Y 753.804,Z 859.31,A -85,B 0,C 180,E1 925.232,E2 925.232} C_VEL
LIN {X 0,Y 753.879,Z 859.31,A -85,B 0,C 180,E1 928.836,E2 928.836} C_VEL
LIN {X 0,Y 753.917,Z 859.31,A -85,B 0,C 180,E1 932.858,E2 932.858} C_VEL
LIN {X 0,Y 754.08,Z 859.31,A -85,B 0,C 180,E1 937.064,E2 937.064} C_VEL
LIN {X 0,Y 753.755,Z 859.31,A -85,B 0,C 180,E1 943.106,E2 943.106} C_VEL
LIN {X 0,Y 753.667,Z 859.31,A -85,B 0,C 180,E1 948.434,E2 948.434} C_VEL
LIN {X 0,Y 753.99,Z 859.31,A -85,B 0,C 180,E1 953.484,E2 953.484} C_VEL
LIN {X 0,Y 753.916,Z 859.31,A -85,B 0,C 180,E1 958.495,E2 958.495} C_VEL
LIN {X 0,Y 754.186,Z 859.31,A -85,B 0,C 180,E1 960.066,E2 960.066} C_VEL
LIN {X 0,Y 755.815,Z 876.391,A -85,B 0,C 180,E1 960.333,E2 960.333} C_VEL
LIN {X 0,Y 755.793,Z 940.152,A -85,B 0,C 180,E1 961.139,E2 961.139} C_VEL
LIN {X 0,Y 755.578,Z 984.686,A -85,B 0,C 180,E1 962.205,E2 962.205} C_VEL
LIN {X 0,Y 755.371,Z 1026.442,A -85,B 0,C 180,E1 963.676,E2 963.676} C_VEL
LIN {X 0,Y 755.095,Z 1067.518,A -85,B 0,C 180,E1 965.629,E2 965.629} C_VEL
LIN {X 0,Y 754.777,Z 1107.449,A -85,B 0,C 180,E1 968.12,E2 968.12} C_VEL
LIN {X 0,Y 754.525,Z 1140.82,A -85,B 0,C 180,E1 970.786,E2 970.786} C_VEL
LIN {X 0,Y 754.287,Z 1171.51,A -85,B 0,C 180,E1 973.922,E2 973.922} C_VEL
LIN {X 0,Y 754.118,Z 1194.791,A -85,B 0,C 180,E1 977.028,E2 977.028} C_VEL
LIN {X 0,Y 754.133,Z 1211.563,A -85,B 0,C 180,E1 979.966,E2 979.966} C_VEL
LIN {X 0,Y 754.058,Z 1224.157,A -85,B 0,C 180,E1 983.075,E2 983.075} C_VEL
LIN {X 0,Y 754.061,Z 1231.66,A -85,B 0,C 180,E1 985.967,E2 985.967} C_VEL
LIN {X 0,Y 754.169,Z 1235.171,A -85,B 0,C 180,E1 988.849,E2 988.849} C_VEL
LIN {X 0,Y 754.223,Z 1234.22,A -85,B 0,C 180,E1 992.303,E2 992.303} C_VEL
LIN {X 0,Y 754.211,Z 1227.633,A -85,B 0,C 180,E1 995.765,E2 995.765} C_VEL
LIN {X 0,Y 754.209,Z 1216.521,A -85,B 0,C 180,E1 998.958,E2 998.958} C_VEL
LIN {X 0,Y 754.223,Z 1198.024,A -85,B 0,C 180,E1 1002.473,E2 1002.473} C_VEL
LIN {X 0,Y 754.304,Z 1175.025,A -85,B 0,C 180,E1 1005.649,E2 1005.649} C_VEL
LIN {X 0,Y 754.491,Z 1147.465,A -85,B 0,C 180,E1 1008.592,E2 1008.592} C_VEL
LIN {X 0,Y 754.715,Z 1115.829,A -85,B 0,C 180,E1 1011.263,E2 1011.263} C_VEL
LIN {X 0,Y 755.02,Z 1079.937,A -85,B 0,C 180,E1 1013.665,E2 1013.665} C_VEL
LIN {X 0,Y 755.341,Z 1037.99,A -85,B 0,C 180,E1 1015.832,E2 1015.832} C_VEL
LIN {X 0,Y 755.632,Z 995.226,A -85,B 0,C 180,E1 1017.466,E2 1017.466} C_VEL
LIN {X 0,Y 755.821,Z 954.352,A -85,B 0,C 180,E1 1018.569,E2 1018.569} C_VEL
LIN {X 0,Y 755.867,Z 911.458,A -85,B 0,C 180,E1 1019.283,E2 1019.283} C_VEL
LIN {X 0,Y 755.32,Z 866.933,A -85,B 0,C 180,E1 1019.79,E2 1019.79} C_VEL
LIN {X 0,Y 754.192,Z 859.31,A -85,B 0,C 180,E1 1019.975,E2 1019.975} C_VEL
LIN {X 0,Y 753.679,Z 859.31,A -85,B 0,C 180,E1 1024.26,E2 1024.26} C_VEL
LIN {X 0,Y 754.138,Z 859.31,A -85,B 0,C 180,E1 1027.07,E2 1027.07} C_VEL
LIN {X 0,Y 754.001,Z 859.31,A -85,B 0,C 180,E1 1033.671,E2 1033.671} C_VEL
LIN {X 0,Y 753.567,Z 859.31,A -85,B 0,C 180,E1 1038.439,E2 1038.439} C_VEL
LIN {X 0,Y 753.605,Z 859.31,A -85,B 0,C 180,E1 1042.909,E2 1042.909} C_VEL
LIN {X 0,Y 753.698,Z 859.31,A -85,B 0,C 180,E1 1047.608,E2 1047.608} C_VEL
LIN {X 0,Y 753.744,Z 859.31,A -85,B 0,C 180,E1 1052.197,E2 1052.197} C_VEL
LIN {X 0,Y 753.834,Z 859.31,A -85,B 0,C 180,E1 1056.3,E2 1056.3} C_VEL
LIN {X 0,Y 753.8,Z 859.31,A -85,B 0,C 180,E1 1060.873,E2 1060.873} C_VEL
LIN {X 0,Y 753.832,Z 859.31,A -85,B 0,C 180,E1 1064.854,E2 1064.854} C_VEL
LIN {X 0,Y 754.08,Z 859.31,A -85,B 0,C 180,E1 1069.942,E2 1069.942} C_VEL
LIN {X 0,Y 753.969,Z 859.31,A -85,B 0,C 180,E1 1074.233,E2 1074.233} C_VEL
LIN {X 0,Y 753.869,Z 859.31,A -85,B 0,C 180,E1 1078.847,E2 1078.847} C_VEL
LIN {X 0,Y 753.908,Z 859.31,A -85,B 0,C 180,E1 1082.302,E2 1082.302} C_VEL
LIN {X 0,Y 753.924,Z 859.31,A -85,B 0,C 180,E1 1085.764,E2 1085.764} C_VEL
LIN {X 0,Y 753.834,Z 859.31,A -85,B 0,C 180,E1 1089.952,E2 1089.952} C_VEL
LIN {X 0,Y 753.757,Z 859.31,A -85,B 0,C 180,E1 1093.954,E2 1093.954} C_VEL
LIN {X 0,Y 753.846,Z 859.31,A -85,B 0,C 180,E1 1097.542,E2 1097.542} C_VEL
LIN {X 0,Y 753.781,Z 859.31,A -85,B 0,C 180,E1 1101.206,E2 1101.206} C_VEL
LIN {X 0,Y 753.749,Z 859.31,A -85,B 0,C 180,E1 1105.224,E2 1105.224} C_VEL
LIN {X 0,Y 753.831,Z 859.31,A -85,B 0,C 180,E1 1108.834,E2 1108.834} C_VEL
LIN {X 0,Y 753.914,Z 859.31,A -85,B 0,C 180,E1 1112.854,E2 1112.854} C_VEL
LIN {X 0,Y 754.109,Z 859.31,A -85,B 0,C 180,E1 1117.058,E2 1117.058} C_VEL
LIN {X 0,Y 753.752,Z 859.31,A -85,B 0,C 180,E1 1123.102,E2 1123.102} C_VEL
LIN {X 0,Y 753.68,Z 859.31,A -85,B 0,C 180,E1 1128.435,E2 1128.435} C_VEL
LIN {X 0,Y 753.97,Z 859.31,A -85,B 0,C 180,E1 1133.481,E2 1133.481} C_VEL
LIN {X 0,Y 753.669,Z 859.31,A -85,B 0,C 180,E1 1138.484,E2 1138.484} C_VEL
LIN {X 0,Y 753.796,Z 859.31,A -85,B 0,C 180,E1 1142.461,E2 1142.461} C_VEL
LIN {X 0,Y 754.067,Z 859.31,A -85,B 0,C 180,E1 1146.099,E2 1146.099} C_VEL
LIN {X 0,Y 755.276,Z 888.688,A -85,B 0,C 180,E1 1146.45,E2 1146.45} C_VEL
LIN {X 0,Y 755.309,Z 968.289,A -85,B 0,C 180,E1 1147.339,E2 1147.339} C_VEL
LIN {X 0,Y 755.171,Z 1007,A -85,B 0,C 180,E1 1148.21,E2 1148.21} C_VEL
LIN {X 0,Y 754.976,Z 1044.372,A -85,B 0,C 180,E1 1149.509,E2 1149.509} C_VEL
LIN {X 0,Y 754.771,Z 1080.417,A -85,B 0,C 180,E1 1151.263,E2 1151.263} C_VEL
LIN {X 0,Y 754.574,Z 1112.818,A -85,B 0,C 180,E1 1153.374,E2 1153.374} C_VEL
LIN {X 0,Y 754.389,Z 1140.625,A -85,B 0,C 180,E1 1155.756,E2 1155.756} C_VEL
LIN {X 0,Y 754.265,Z 1164.141,A -85,B 0,C 180,E1 1158.411,E2 1158.411} C_VEL
LIN {X 0,Y 754.161,Z 1181.488,A -85,B 0,C 180,E1 1161.042,E2 1161.042} C_VEL
LIN {X 0,Y 754.131,Z 1194.78,A -85,B 0,C 180,E1 1163.942,E2 1163.942} C_VEL
LIN {X 0,Y 754.103,Z 1202.02,A -85,B 0,C 180,E1 1166.544,E2 1166.544} C_VEL
LIN {X 0,Y 754.088,Z 1205.12,A -85,B 0,C 180,E1 1168.849,E2 1168.849} C_VEL
LIN {X 0,Y 754.139,Z 1205.041,A -85,B 0,C 180,E1 1171.151,E2 1171.151} C_VEL
LIN {X 0,Y 754.163,Z 1200.601,A -85,B 0,C 180,E1 1174.033,E2 1174.033} C_VEL
LIN {X 0,Y 754.194,Z 1189.719,A -85,B 0,C 180,E1 1177.214,E2 1177.214} C_VEL
LIN {X 0,Y 754.266,Z 1174.037,A -85,B 0,C 180,E1 1180.097,E2 1180.097} C_VEL
LIN {X 0,Y 754.355,Z 1152.666,A -85,B 0,C 180,E1 1182.888,E2 1182.888} C_VEL
LIN {X 0,Y 754.451,Z 1127.503,A -85,B 0,C 180,E1 1185.354,E2 1185.354} C_VEL
LIN {X 0,Y 754.627,Z 1098.617,A -85,B 0,C 180,E1 1187.53,E2 1187.53} C_VEL
LIN {X 0,Y 754.807,Z 1065.756,A -85,B 0,C 180,E1 1189.426,E2 1189.426} C_VEL
LIN {X 0,Y 755.028,Z 1030.103,A -85,B 0,C 180,E1 1190.954,E2 1190.954} C_VEL
LIN {X 0,Y 755.183,Z 991.675,A -85,B 0,C 180,E1 1192.1,E2 1192.1} C_VEL
LIN {X 0,Y 755.246,Z 953.911,A -85,B 0,C 180,E1 1192.784,E2 1192.784} C_VEL
LIN {X 0,Y 754.532,Z 861.91,A -85,B 0,C 180,E1 1193.757,E2 1193.757} C_VEL
LIN {X 0,Y 754.052,Z 859.31,A -85,B 0,C 180,E1 1193.886,E2 1193.886} C_VEL
LIN {X 0,Y 753.871,Z 859.31,A -85,B 0,C 180,E1 1198.843,E2 1198.843} C_VEL
LIN {X 0,Y 753.945,Z 859.31,A -85,B 0,C 180,E1 1202.864,E2 1202.864} C_VEL
LIN {X 0,Y 754.118,Z 859.31,A -85,B 0,C 180,E1 1207.071,E2 1207.071} C_VEL
LIN {X 0,Y 753.708,Z 859.31,A -85,B 0,C 180,E1 1213.122,E2 1213.122} C_VEL
LIN {X 0,Y 753.691,Z 859.31,A -85,B 0,C 180,E1 1218.451,E2 1218.451} C_VEL
LIN {X 0,Y 753.935,Z 859.31,A -85,B 0,C 180,E1 1223.508,E2 1223.508} C_VEL
LIN {X 0,Y 753.669,Z 859.31,A -85,B 0,C 180,E1 1228.495,E2 1228.495} C_VEL
LIN {X 0,Y 753.836,Z 859.31,A -85,B 0,C 180,E1 1232.472,E2 1232.472} C_VEL
LIN {X 0,Y 753.836,Z 859.31,A -85,B 0,C 180,E1 1237.555,E2 1237.555} C_VEL
LIN {X 0,Y 753.619,Z 859.31,A -85,B 0,C 180,E1 1241.24,E2 1241.24} C_VEL
LIN {X 0,Y 753.891,Z 859.31,A -85,B 0,C 180,E1 1246.048,E2 1246.048} C_VEL
LIN {X 0,Y 753.902,Z 859.31,A -85,B 0,C 180,E1 1250.751,E2 1250.751} C_VEL
LIN {X 0,Y 753.937,Z 859.31,A -85,B 0,C 180,E1 1254.612,E2 1254.612} C_VEL
LIN {X 0,Y 754.025,Z 859.31,A -85,B 0,C 180,E1 1257.199,E2 1257.199} C_VEL
LIN {X 0,Y 752.759,Z 859.31,A -85,B 0,C 180,E1 1257.857,E2 1257.857} C_VEL
LIN {X 0,Y 746.126,Z 859.31,A -85,B 0,C 180,E1 1259.643,E2 1259.643} C_VEL
LIN {X 0,Y 746.058,Z 859.31,A -85,B 0,C 180,E1 1259.811,E2 1259.811} C_VEL
LIN {X 0,Y 746.264,Z 859.31,A -85,B 0,C 180,E1 1264.659,E2 1264.659} C_VEL
LIN {X 0,Y 746.011,Z 859.31,A -85,B 0,C 180,E1 1269.351,E2 1269.351} C_VEL
LIN {X 0,Y 745.853,Z 859.31,A -85,B 0,C 180,E1 1274.108,E2 1274.108} C_VEL
LIN {X 0,Y 745.956,Z 859.31,A -85,B 0,C 180,E1 1277.737,E2 1277.737} C_VEL
LIN {X 0,Y 745.938,Z 859.31,A -85,B 0,C 180,E1 1281.443,E2 1281.443} C_VEL
LIN {X 0,Y 745.926,Z 859.31,A -85,B 0,C 180,E1 1285.246,E2 1285.246} C_VEL
LIN {X 0,Y 745.898,Z 859.31,A -85,B 0,C 180,E1 1289.174,E2 1289.174} C_VEL
LIN {X 0,Y 745.828,Z 859.31,A -85,B 0,C 180,E1 1293.592,E2 1293.592} C_VEL
LIN {X 0,Y 745.984,Z 859.31,A -85,B 0,C 180,E1 1297.609,E2 1297.609} C_VEL
LIN {X 0,Y 745.85,Z 859.31,A -85,B 0,C 180,E1 1302.997,E2 1302.997} C_VEL
LIN {X 0,Y 745.839,Z 859.31,A -85,B 0,C 180,E1 1307.898,E2 1307.898} C_VEL
LIN {X 0,Y 746.071,Z 859.31,A -85,B 0,C 180,E1 1312.46,E2 1312.46} C_VEL
LIN {X 0,Y 746.022,Z 859.31,A -85,B 0,C 180,E1 1318.122,E2 1318.122} C_VEL
LIN {X 0,Y 746.223,Z 860.078,A -85,B 0,C 180,E1 1319.735,E2 1319.735} C_VEL
LIN {X 0,Y 748.947,Z 873.887,A -85,B 0,C 180,E1 1320.006,E2 1320.006} C_VEL
LIN {X 0,Y 748.867,Z 939.48,A -85,B 0,C 180,E1 1320.836,E2 1320.836} C_VEL
LIN {X 0,Y 748.494,Z 982.824,A -85,B 0,C 180,E1 1321.864,E2 1321.864} C_VEL
LIN {X 0,Y 748.147,Z 1025.167,A -85,B 0,C 180,E1 1323.347,E2 1323.347} C_VEL
LIN {X 0,Y 747.728,Z 1067.424,A -85,B 0,C 180,E1 1325.368,E2 1325.368} C_VEL
LIN {X 0,Y 747.222,Z 1107.447,A -85,B 0,C 180,E1 1327.887,E2 1327.887} C_VEL
LIN {X 0,Y 746.84,Z 1142.108,A -85,B 0,C 180,E1 1330.699,E2 1330.699} C_VEL
LIN {X 0,Y 746.501,Z 1171.882,A -85,B 0,C 180,E1 1333.793,E2 1333.793} C_VEL
LIN {X 0,Y 746.275,Z 1195.565,A -85,B 0,C 180,E1 1337.007,E2 1337.007} C_VEL
LIN {X 0,Y 746.253,Z 1211.564,A -85,B 0,C 180,E1 1339.859,E2 1339.859} C_VEL
LIN {X 0,Y 746.184,Z 1224.157,A -85,B 0,C 180,E1 1343.001,E2 1343.001} C_VEL
LIN {X 0,Y 746.188,Z 1231.661,A -85,B 0,C 180,E1 1345.924,E2 1345.924} C_VEL
LIN {X 0,Y 746.266,Z 1235.171,A -85,B 0,C 180,E1 1348.836,E2 1348.836} C_VEL
LIN {X 0,Y 746.317,Z 1234.22,A -85,B 0,C 180,E1 1352.327,E2 1352.327} C_VEL
LIN {X 0,Y 746.286,Z 1227.405,A -85,B 0,C 180,E1 1355.912,E2 1355.912} C_VEL
LIN {X 0,Y 746.262,Z 1215.178,A -85,B 0,C 180,E1 1359.348,E2 1359.348} C_VEL
LIN {X 0,Y 746.348,Z 1198.025,A -85,B 0,C 180,E1 1362.606,E2 1362.606} C_VEL
LIN {X 0,Y 746.476,Z 1174.324,A -85,B 0,C 180,E1 1365.905,E2 1365.905} C_VEL
LIN {X 0,Y 746.762,Z 1147.466,A -85,B 0,C 180,E1 1368.791,E2 1368.791} C_VEL
LIN {X 0,Y 747.14,Z 1115.83,A -85,B 0,C 180,E1 1371.489,E2 1371.489} C_VEL
LIN {X 0,Y 747.615,Z 1078.412,A -85,B 0,C 180,E1 1374.002,E2 1374.002} C_VEL
LIN {X 0,Y 748.079,Z 1037.847,A -85,B 0,C 180,E1 1376.109,E2 1376.109} C_VEL
LIN {X 0,Y 748.536,Z 995.23,A -85,B 0,C 180,E1 1377.749,E2 1377.749} C_VEL
LIN {X 0,Y 748.855,Z 955.085,A -85,B 0,C 180,E1 1378.845,E2 1378.845} C_VEL
LIN {X 0,Y 748.977,Z 912.164,A -85,B 0,C 180,E1 1379.57,E2 1379.57} C_VEL
LIN {X 0,Y 748.238,Z 867.961,A -85,B 0,C 180,E1 1380.089,E2 1380.089} C_VEL
LIN {X 0,Y 746.195,Z 859.31,A -85,B 0,C 180,E1 1380.312,E2 1380.312} C_VEL
LIN {X 0,Y 745.861,Z 859.31,A -85,B 0,C 180,E1 1385.664,E2 1385.664} C_VEL
LIN {X 0,Y 745.667,Z 859.31,A -85,B 0,C 180,E1 1389.463,E2 1389.463} C_VEL
LIN {X 0,Y 746.101,Z 859.31,A -85,B 0,C 180,E1 1393.671,E2 1393.671} C_VEL
LIN {X 0,Y 745.686,Z 859.31,A -85,B 0,C 180,E1 1398.752,E2 1398.752} C_VEL
LIN {X 0,Y 745.715,Z 859.31,A -85,B 0,C 180,E1 1402.449,E2 1402.449} C_VEL
LIN {X 0,Y 745.756,Z 859.31,A -85,B 0,C 180,E1 1406.736,E2 1406.736} C_VEL
LIN {X 0,Y 745.819,Z 859.31,A -85,B 0,C 180,E1 1410.884,E2 1410.884} C_VEL
LIN {X 0,Y 746.024,Z 859.31,A -85,B 0,C 180,E1 1414.757,E2 1414.757} C_VEL
LIN {X 0,Y 745.914,Z 859.31,A -85,B 0,C 180,E1 1419.142,E2 1419.142} C_VEL
LIN {X 0,Y 745.98,Z 859.31,A -85,B 0,C 180,E1 1423.481,E2 1423.481} C_VEL
LIN {X 0,Y 745.811,Z 859.31,A -85,B 0,C 180,E1 1428.279,E2 1428.279} C_VEL
LIN {X 0,Y 746.15,Z 859.31,A -85,B 0,C 180,E1 1433.001,E2 1433.001} C_VEL
LIN {X 0,Y 746.169,Z 859.31,A -85,B 0,C 180,E1 1437.671,E2 1437.671} C_VEL
LIN {X 0,Y 746.007,Z 859.31,A -85,B 0,C 180,E1 1442.326,E2 1442.326} C_VEL
LIN {X 0,Y 746.013,Z 859.31,A -85,B 0,C 180,E1 1445.826,E2 1445.826} C_VEL
LIN {X 0,Y 745.905,Z 859.31,A -85,B 0,C 180,E1 1450.53,E2 1450.53} C_VEL
LIN {X 0,Y 746.019,Z 859.31,A -85,B 0,C 180,E1 1455.305,E2 1455.305} C_VEL
LIN {X 0,Y 746.046,Z 859.31,A -85,B 0,C 180,E1 1460.192,E2 1460.192} C_VEL
LIN {X 0,Y 745.872,Z 859.31,A -85,B 0,C 180,E1 1465.245,E2 1465.245} C_VEL
LIN {X 0,Y 745.869,Z 859.31,A -85,B 0,C 180,E1 1469.171,E2 1469.171} C_VEL
LIN {X 0,Y 745.824,Z 859.31,A -85,B 0,C 180,E1 1473.592,E2 1473.592} C_VEL
LIN {X 0,Y 746.014,Z 859.31,A -85,B 0,C 180,E1 1477.612,E2 1477.612} C_VEL
LIN {X 0,Y 745.846,Z 859.31,A -85,B 0,C 180,E1 1482.997,E2 1482.997} C_VEL
LIN {X 0,Y 745.849,Z 859.31,A -85,B 0,C 180,E1 1487.899,E2 1487.899} C_VEL
LIN {X 0,Y 746.067,Z 859.31,A -85,B 0,C 180,E1 1492.46,E2 1492.46} C_VEL
LIN {X 0,Y 745.915,Z 859.31,A -85,B 0,C 180,E1 1496.736,E2 1496.736} C_VEL
LIN {X 0,Y 745.952,Z 859.31,A -85,B 0,C 180,E1 1502.147,E2 1502.147} C_VEL
LIN {X 0,Y 746.181,Z 859.31,A -85,B 0,C 180,E1 1505.822,E2 1505.822} C_VEL
LIN {X 0,Y 748.037,Z 875.982,A -85,B 0,C 180,E1 1506.078,E2 1506.078} C_VEL
LIN {X 0,Y 748.017,Z 968.391,A -85,B 0,C 180,E1 1507.107,E2 1507.107} C_VEL
LIN {X 0,Y 747.788,Z 1006.985,A -85,B 0,C 180,E1 1507.983,E2 1507.983} C_VEL
LIN {X 0,Y 747.483,Z 1044.511,A -85,B 0,C 180,E1 1509.3,E2 1509.3} C_VEL
LIN {X 0,Y 747.178,Z 1080.411,A -85,B 0,C 180,E1 1511.066,E2 1511.066} C_VEL
LIN {X 0,Y 746.876,Z 1113.161,A -85,B 0,C 180,E1 1513.224,E2 1513.224} C_VEL
LIN {X 0,Y 746.581,Z 1142.089,A -85,B 0,C 180,E1 1515.754,E2 1515.754} C_VEL
LIN {X 0,Y 746.425,Z 1165.232,A -85,B 0,C 180,E1 1518.436,E2 1518.436} C_VEL
LIN {X 0,Y 746.289,Z 1183.025,A -85,B 0,C 180,E1 1521.241,E2 1521.241} C_VEL
LIN {X 0,Y 746.247,Z 1195.75,A -85,B 0,C 180,E1 1524.173,E2 1524.173} C_VEL
LIN {X 0,Y 746.204,Z 1202.019,A -85,B 0,C 180,E1 1526.508,E2 1526.508} C_VEL
LIN {X 0,Y 746.189,Z 1205.12,A -85,B 0,C 180,E1 1528.837,E2 1528.837} C_VEL
LIN {X 0,Y 746.238,Z 1205.042,A -85,B 0,C 180,E1 1531.164,E2 1531.164} C_VEL
LIN {X 0,Y 746.279,Z 1200.603,A -85,B 0,C 180,E1 1534.075,E2 1534.075} C_VEL
LIN {X 0,Y 746.333,Z 1189.721,A -85,B 0,C 180,E1 1537.29,E2 1537.29} C_VEL
LIN {X 0,Y 746.391,Z 1174.041,A -85,B 0,C 180,E1 1540.205,E2 1540.205} C_VEL
LIN {X 0,Y 746.534,Z 1153.783,A -85,B 0,C 180,E1 1542.902,E2 1542.902} C_VEL
LIN {X 0,Y 746.691,Z 1128.125,A -85,B 0,C 180,E1 1545.464,E2 1545.464} C_VEL
LIN {X 0,Y 747.027,Z 1097.484,A -85,B 0,C 180,E1 1547.79,E2 1547.79} C_VEL
LIN {X 0,Y 747.276,Z 1063.594,A -85,B 0,C 180,E1 1549.74,E2 1549.74} C_VEL
LIN {X 0,Y 747.567,Z 1026.182,A -85,B 0,C 180,E1 1551.318,E2 1551.318} C_VEL
LIN {X 0,Y 747.915,Z 985.134,A -85,B 0,C 180,E1 1552.483,E2 1552.483} C_VEL
LIN {X 0,Y 748.005,Z 943.836,A -85,B 0,C 180,E1 1553.137,E2 1553.137} C_VEL
LIN {X 0,Y 747.247,Z 863.407,A -85,B 0,C 180,E1 1553.988,E2 1553.988} C_VEL
LIN {X 0,Y 746.045,Z 859.31,A -85,B 0,C 180,E1 1554.099,E2 1554.099} C_VEL
LIN {X 0,Y 745.9,Z 859.31,A -85,B 0,C 180,E1 1559.18,E2 1559.18} C_VEL
LIN {X 0,Y 745.864,Z 859.31,A -85,B 0,C 180,E1 1563.623,E2 1563.623} C_VEL
LIN {X 0,Y 746.025,Z 859.31,A -85,B 0,C 180,E1 1567.635,E2 1567.635} C_VEL
LIN {X 0,Y 745.811,Z 859.31,A -85,B 0,C 180,E1 1573.013,E2 1573.013} C_VEL
LIN {X 0,Y 745.861,Z 859.31,A -85,B 0,C 180,E1 1577.916,E2 1577.916} C_VEL
LIN {X 0,Y 746.049,Z 859.31,A -85,B 0,C 180,E1 1582.473,E2 1582.473} C_VEL
LIN {X 0,Y 745.912,Z 859.31,A -85,B 0,C 180,E1 1586.748,E2 1586.748} C_VEL
LIN {X 0,Y 745.972,Z 859.31,A -85,B 0,C 180,E1 1592.157,E2 1592.157} C_VEL
LIN {X 0,Y 745.953,Z 859.31,A -85,B 0,C 180,E1 1597.305,E2 1597.305} C_VEL
LIN {X 0,Y 745.813,Z 859.31,A -85,B 0,C 180,E1 1601.037,E2 1601.037} C_VEL
LIN {X 0,Y 745.948,Z 859.31,A -85,B 0,C 180,E1 1605.897,E2 1605.897} C_VEL
LIN {X 0,Y 746.038,Z 859.31,A -85,B 0,C 180,E1 1610.653,E2 1610.653} C_VEL
LIN {X 0,Y 746.085,Z 859.31,A -85,B 0,C 180,E1 1614.377,E2 1614.377} C_VEL
LIN {X 0,Y 746.003,Z 859.31,A -85,B 0,C 180,E1 1618.838,E2 1618.838} C_VEL
LIN {X 0,Y 746.058,Z 859.31,A -85,B 0,C 180,E1 1619.811,E2 1619.811} C_VEL
LIN {X 0,Y 743.614,Z 859.31,A -85,B 0,C 180,E1 1620.803,E2 1620.803} C_VEL
LIN {X 0,Y 738.206,Z 859.31,A -85,B 0,C 180,E1 1622.282,E2 1622.282} C_VEL
LIN {X 0,Y 738.101,Z 859.31,A -85,B 0,C 180,E1 1622.453,E2 1622.453} C_VEL
LIN {X 0,Y 738.106,Z 859.31,A -85,B 0,C 180,E1 1625.892,E2 1625.892} C_VEL
LIN {X 0,Y 737.987,Z 859.31,A -85,B 0,C 180,E1 1630.648,E2 1630.648} C_VEL
LIN {X 0,Y 738.128,Z 859.31,A -85,B 0,C 180,E1 1635.476,E2 1635.476} C_VEL
LIN {X 0,Y 738.164,Z 859.31,A -85,B 0,C 180,E1 1640.421,E2 1640.421} C_VEL
LIN {X 0,Y 737.98,Z 859.31,A -85,B 0,C 180,E1 1645.538,E2 1645.538} C_VEL
LIN {X 0,Y 737.926,Z 859.31,A -85,B 0,C 180,E1 1650.407,E2 1650.407} C_VEL
LIN {X 0,Y 737.846,Z 859.31,A -85,B 0,C 180,E1 1655.093,E2 1655.093} C_VEL
LIN {X 0,Y 737.723,Z 859.31,A -85,B 0,C 180,E1 1659.539,E2 1659.539} C_VEL
LIN {X 0,Y 737.79,Z 859.31,A -85,B 0,C 180,E1 1664.041,E2 1664.041} C_VEL
LIN {X 0,Y 737.783,Z 859.31,A -85,B 0,C 180,E1 1668.911,E2 1668.911} C_VEL
LIN {X 0,Y 738.081,Z 859.31,A -85,B 0,C 180,E1 1673.46,E2 1673.46} C_VEL
LIN {X 0,Y 738.065,Z 859.31,A -85,B 0,C 180,E1 1677.738,E2 1677.738} C_VEL
LIN {X 0,Y 738.229,Z 859.837,A -85,B 0,C 180,E1 1679.369,E2 1679.369} C_VEL
LIN {X 0,Y 742.026,Z 872.065,A -85,B 0,C 180,E1 1679.677,E2 1679.677} C_VEL
LIN {X 0,Y 741.953,Z 939.482,A -85,B 0,C 180,E1 1680.537,E2 1680.537} C_VEL
LIN {X 0,Y 741.442,Z 983.637,A -85,B 0,C 180,E1 1681.596,E2 1681.596} C_VEL
LIN {X 0,Y 740.917,Z 1026.291,A -85,B 0,C 180,E1 1683.114,E2 1683.114} C_VEL
LIN {X 0,Y 740.341,Z 1067.515,A -85,B 0,C 180,E1 1685.111,E2 1685.111} C_VEL
LIN {X 0,Y 739.715,Z 1106.772,A -85,B 0,C 180,E1 1687.6,E2 1687.6} C_VEL
LIN {X 0,Y 739.202,Z 1140.921,A -85,B 0,C 180,E1 1690.38,E2 1690.38} C_VEL
LIN {X 0,Y 738.713,Z 1170.559,A -85,B 0,C 180,E1 1693.464,E2 1693.464} C_VEL
LIN {X 0,Y 738.442,Z 1194.173,A -85,B 0,C 180,E1 1696.653,E2 1696.653} C_VEL
LIN {X 0,Y 738.372,Z 1211.523,A -85,B 0,C 180,E1 1699.74,E2 1699.74} C_VEL
LIN {X 0,Y 738.294,Z 1224.157,A -85,B 0,C 180,E1 1702.926,E2 1702.926} C_VEL
LIN {X 0,Y 738.292,Z 1231.661,A -85,B 0,C 180,E1 1705.88,E2 1705.88} C_VEL
LIN {X 0,Y 738.364,Z 1235.17,A -85,B 0,C 180,E1 1708.824,E2 1708.824} C_VEL
LIN {X 0,Y 738.427,Z 1234.22,A -85,B 0,C 180,E1 1712.352,E2 1712.352} C_VEL
LIN {X 0,Y 738.414,Z 1227.634,A -85,B 0,C 180,E1 1715.889,E2 1715.889} C_VEL
LIN {X 0,Y 738.409,Z 1216.52,A -85,B 0,C 180,E1 1719.151,E2 1719.151} C_VEL
LIN {X 0,Y 738.48,Z 1198.026,A -85,B 0,C 180,E1 1722.743,E2 1722.743} C_VEL
LIN {X 0,Y 738.669,Z 1175.541,A -85,B 0,C 180,E1 1725.924,E2 1725.924} C_VEL
LIN {X 0,Y 739.048,Z 1149.078,A -85,B 0,C 180,E1 1728.84,E2 1728.84} C_VEL
LIN {X 0,Y 739.557,Z 1116.877,A -85,B 0,C 180,E1 1731.642,E2 1731.642} C_VEL
LIN {X 0,Y 740.179,Z 1079.943,A -85,B 0,C 180,E1 1734.169,E2 1734.169} C_VEL
LIN {X 0,Y 740.824,Z 1038.792,A -85,B 0,C 180,E1 1736.338,E2 1736.338} C_VEL
LIN {X 0,Y 741.424,Z 996.602,A -85,B 0,C 180,E1 1737.991,E2 1737.991} C_VEL
LIN {X 0,Y 741.918,Z 955.673,A -85,B 0,C 180,E1 1739.128,E2 1739.128} C_VEL
LIN {X 0,Y 742.126,Z 910.19,A -85,B 0,C 180,E1 1739.897,E2 1739.897} C_VEL
LIN {X 0,Y 741.404,Z 869.535,A -85,B 0,C 180,E1 1740.379,E2 1740.379} C_VEL
LIN {X 0,Y 738.267,Z 859.31,A -85,B 0,C 180,E1 1740.66,E2 1740.66} C_VEL
LIN {X 0,Y 738.028,Z 859.31,A -85,B 0,C 180,E1 1746.542,E2 1746.542} C_VEL
LIN {X 0,Y 738.082,Z 859.31,A -85,B 0,C 180,E1 1752.648,E2 1752.648} C_VEL
LIN {X 0,Y 737.772,Z 859.31,A -85,B 0,C 180,E1 1757.342,E2 1757.342} C_VEL
LIN {X 0,Y 737.826,Z 859.31,A -85,B 0,C 180,E1 1761.977,E2 1761.977} C_VEL
LIN {X 0,Y 737.878,Z 859.31,A -85,B 0,C 180,E1 1766.334,E2 1766.334} C_VEL
LIN {X 0,Y 737.916,Z 859.31,A -85,B 0,C 180,E1 1770.48,E2 1770.48} C_VEL
LIN {X 0,Y 738.133,Z 859.31,A -85,B 0,C 180,E1 1774.59,E2 1774.59} C_VEL
LIN {X 0,Y 738.115,Z 859.31,A -85,B 0,C 180,E1 1778.318,E2 1778.318} C_VEL
LIN {X 0,Y 738.099,Z 859.31,A -85,B 0,C 180,E1 1783.3,E2 1783.3} C_VEL
LIN {X 0,Y 737.911,Z 859.31,A -85,B 0,C 180,E1 1788.152,E2 1788.152} C_VEL
LIN {X 0,Y 738.223,Z 859.31,A -85,B 0,C 180,E1 1792.926,E2 1792.926} C_VEL
LIN {X 0,Y 738.268,Z 859.31,A -85,B 0,C 180,E1 1797.646,E2 1797.646} C_VEL
LIN {X 0,Y 738.116,Z 859.31,A -85,B 0,C 180,E1 1802.351,E2 1802.351} C_VEL
LIN {X 0,Y 738.102,Z 859.31,A -85,B 0,C 180,E1 1805.888,E2 1805.888} C_VEL
LIN {X 0,Y 738.033,Z 859.31,A -85,B 0,C 180,E1 1810.644,E2 1810.644} C_VEL
LIN {X 0,Y 738.124,Z 859.31,A -85,B 0,C 180,E1 1815.473,E2 1815.473} C_VEL
LIN {X 0,Y 738.107,Z 859.31,A -85,B 0,C 180,E1 1820.419,E2 1820.419} C_VEL
LIN {X 0,Y 737.935,Z 859.31,A -85,B 0,C 180,E1 1825.536,E2 1825.536} C_VEL
LIN {X 0,Y 737.888,Z 859.31,A -85,B 0,C 180,E1 1830.403,E2 1830.403} C_VEL
LIN {X 0,Y 737.862,Z 859.31,A -85,B 0,C 180,E1 1835.088,E2 1835.088} C_VEL
LIN {X 0,Y 737.742,Z 859.31,A -85,B 0,C 180,E1 1839.534,E2 1839.534} C_VEL
LIN {X 0,Y 737.796,Z 859.31,A -85,B 0,C 180,E1 1844.042,E2 1844.042} C_VEL
LIN {X 0,Y 737.822,Z 859.31,A -85,B 0,C 180,E1 1848.914,E2 1848.914} C_VEL
LIN {X 0,Y 738.065,Z 859.31,A -85,B 0,C 180,E1 1853.46,E2 1853.46} C_VEL
LIN {X 0,Y 737.924,Z 859.31,A -85,B 0,C 180,E1 1857.731,E2 1857.731} C_VEL
LIN {X 0,Y 738.019,Z 859.31,A -85,B 0,C 180,E1 1861.959,E2 1861.959} C_VEL
LIN {X 0,Y 738.181,Z 859.31,A -85,B 0,C 180,E1 1865.551,E2 1865.551} C_VEL
LIN {X 0,Y 740.824,Z 873.383,A -85,B 0,C 180,E1 1865.804,E2 1865.804} C_VEL
LIN {X 0,Y 740.729,Z 966.659,A -85,B 0,C 180,E1 1866.842,E2 1866.842} C_VEL
LIN {X 0,Y 740.432,Z 1005.578,A -85,B 0,C 180,E1 1867.713,E2 1867.713} C_VEL
LIN {X 0,Y 740.068,Z 1042.195,A -85,B 0,C 180,E1 1868.987,E2 1868.987} C_VEL
LIN {X 0,Y 739.595,Z 1077.484,A -85,B 0,C 180,E1 1870.699,E2 1870.699} C_VEL
LIN {X 0,Y 739.189,Z 1110.293,A -85,B 0,C 180,E1 1872.832,E2 1872.832} C_VEL
LIN {X 0,Y 738.781,Z 1139.129,A -85,B 0,C 180,E1 1875.296,E2 1875.296} C_VEL
LIN {X 0,Y 738.57,Z 1163.042,A -85,B 0,C 180,E1 1878.011,E2 1878.011} C_VEL
LIN {X 0,Y 738.406,Z 1181.484,A -85,B 0,C 180,E1 1880.849,E2 1880.849} C_VEL
LIN {X 0,Y 738.339,Z 1194.787,A -85,B 0,C 180,E1 1883.815,E2 1883.815} C_VEL
LIN {X 0,Y 738.334,Z 1202.019,A -85,B 0,C 180,E1 1886.47,E2 1886.47} C_VEL
LIN {X 0,Y 738.289,Z 1205.12,A -85,B 0,C 180,E1 1888.824,E2 1888.824} C_VEL
LIN {X 0,Y 738.337,Z 1205.042,A -85,B 0,C 180,E1 1891.176,E2 1891.176} C_VEL
LIN {X 0,Y 738.377,Z 1200.605,A -85,B 0,C 180,E1 1894.119,E2 1894.119} C_VEL
LIN {X 0,Y 738.469,Z 1189.723,A -85,B 0,C 180,E1 1897.368,E2 1897.368} C_VEL
LIN {X 0,Y 738.526,Z 1174.15,A -85,B 0,C 180,E1 1900.299,E2 1900.299} C_VEL
LIN {X 0,Y 738.693,Z 1153.786,A -85,B 0,C 180,E1 1903.041,E2 1903.041} C_VEL
LIN {X 0,Y 738.956,Z 1128.507,A -85,B 0,C 180,E1 1905.598,E2 1905.598} C_VEL
LIN {X 0,Y 739.371,Z 1098.636,A -85,B 0,C 180,E1 1907.904,E2 1907.904} C_VEL
LIN {X 0,Y 739.706,Z 1065.412,A -85,B 0,C 180,E1 1909.858,E2 1909.858} C_VEL
LIN {X 0,Y 740.164,Z 1029.508,A -85,B 0,C 180,E1 1911.419,E2 1911.419} C_VEL
LIN {X 0,Y 740.515,Z 991.723,A -85,B 0,C 180,E1 1912.562,E2 1912.562} C_VEL
LIN {X 0,Y 740.711,Z 952.868,A -85,B 0,C 180,E1 1913.271,E2 1913.271} C_VEL
LIN {X 0,Y 739.948,Z 865.514,A -85,B 0,C 180,E1 1914.218,E2 1914.218} C_VEL
LIN {X 0,Y 738.041,Z 859.31,A -85,B 0,C 180,E1 1914.387,E2 1914.387} C_VEL
LIN {X 0,Y 737.934,Z 859.31,A -85,B 0,C 180,E1 1919.526,E2 1919.526} C_VEL
LIN {X 0,Y 737.954,Z 859.31,A -85,B 0,C 180,E1 1923.67,E2 1923.67} C_VEL
LIN {X 0,Y 737.878,Z 859.31,A -85,B 0,C 180,E1 1928.728,E2 1928.728} C_VEL
LIN {X 0,Y 737.938,Z 859.31,A -85,B 0,C 180,E1 1932.659,E2 1932.659} C_VEL
LIN {X 0,Y 737.962,Z 859.31,A -85,B 0,C 180,E1 1937.664,E2 1937.664} C_VEL
LIN {X 0,Y 738.05,Z 859.31,A -85,B 0,C 180,E1 1943.472,E2 1943.472} C_VEL
LIN {X 0,Y 737.929,Z 859.31,A -85,B 0,C 180,E1 1947.743,E2 1947.743} C_VEL
LIN {X 0,Y 737.983,Z 859.31,A -85,B 0,C 180,E1 1953.155,E2 1953.155} C_VEL
LIN {X 0,Y 738.031,Z 859.31,A -85,B 0,C 180,E1 1957.507,E2 1957.507} C_VEL
LIN {X 0,Y 737.936,Z 859.31,A -85,B 0,C 180,E1 1960.835,E2 1960.835} C_VEL
LIN {X 0,Y 738.01,Z 859.31,A -85,B 0,C 180,E1 1965.742,E2 1965.742} C_VEL
LIN {X 0,Y 738.142,Z 859.31,A -85,B 0,C 180,E1 1970.552,E2 1970.552} C_VEL
LIN {X 0,Y 738.084,Z 859.31,A -85,B 0,C 180,E1 1975.292,E2 1975.292} C_VEL
LIN {X 0,Y 738.198,Z 859.31,A -85,B 0,C 180,E1 1980.002,E2 1980.002} C_VEL
LIN {X 0,Y 738.101,Z 859.31,A -85,B 0,C 180,E1 1982.453,E2 1982.453} C_VEL
LIN {X 0,Y 734.288,Z 859.31,A -85,B 0,C 180,E1 1983.778,E2 1983.778} C_VEL
LIN {X 0,Y 730.354,Z 859.31,A -85,B 0,C 180,E1 1985.117,E2 1985.117} C_VEL
LIN {X 0,Y 730.173,Z 859.31,A -85,B 0,C 180,E1 1989.556,E2 1989.556} C_VEL
LIN {X 0,Y 730.075,Z 859.31,A -85,B 0,C 180,E1 1994.42,E2 1994.42} C_VEL
LIN {X 0,Y 730.233,Z 859.31,A -85,B 0,C 180,E1 1999.387,E2 1999.387} C_VEL
LIN {X 0,Y 730.19,Z 859.31,A -85,B 0,C 180,E1 2004.517,E2 2004.517} C_VEL
LIN {X 0,Y 730.02,Z 859.31,A -85,B 0,C 180,E1 2009.872,E2 2009.872} C_VEL
LIN {X 0,Y 729.98,Z 859.31,A -85,B 0,C 180,E1 2014.08,E2 2014.08} C_VEL
LIN {X 0,Y 729.947,Z 859.31,A -85,B 0,C 180,E1 2018.508,E2 2018.508} C_VEL
LIN {X 0,Y 729.916,Z 859.31,A -85,B 0,C 180,E1 2023.398,E2 2023.398} C_VEL
LIN {X 0,Y 729.915,Z 859.31,A -85,B 0,C 180,E1 2028.37,E2 2028.37} C_VEL
LIN {X 0,Y 730.166,Z 859.31,A -85,B 0,C 180,E1 2032.999,E2 2032.999} C_VEL
LIN {X 0,Y 730.192,Z 859.31,A -85,B 0,C 180,E1 2038.281,E2 2038.281} C_VEL
LIN {X 0,Y 730.265,Z 859.31,A -85,B 0,C 180,E1 2038.971,E2 2038.971} C_VEL
LIN {X 0,Y 735.176,Z 873.561,A -85,B 0,C 180,E1 2039.381,E2 2039.381} C_VEL
LIN {X 0,Y 735.056,Z 940.146,A -85,B 0,C 180,E1 2040.244,E2 2040.244} C_VEL
LIN {X 0,Y 734.407,Z 984.714,A -85,B 0,C 180,E1 2041.331,E2 2041.331} C_VEL
LIN {X 0,Y 733.72,Z 1027.046,A -85,B 0,C 180,E1 2042.862,E2 2042.862} C_VEL
LIN {X 0,Y 732.969,Z 1067.521,A -85,B 0,C 180,E1 2044.844,E2 2044.844} C_VEL
LIN {X 0,Y 732.175,Z 1106.08,A -85,B 0,C 180,E1 2047.306,E2 2047.306} C_VEL
LIN {X 0,Y 731.522,Z 1141.251,A -85,B 0,C 180,E1 2050.196,E2 2050.196} C_VEL
LIN {X 0,Y 730.92,Z 1171.881,A -85,B 0,C 180,E1 2053.438,E2 2053.438} C_VEL
LIN {X 0,Y 730.591,Z 1196.14,A -85,B 0,C 180,E1 2056.812,E2 2056.812} C_VEL
LIN {X 0,Y 730.496,Z 1212.686,A -85,B 0,C 180,E1 2059.889,E2 2059.889} C_VEL
LIN {X 0,Y 730.412,Z 1224.157,A -85,B 0,C 180,E1 2062.849,E2 2062.849} C_VEL
LIN {X 0,Y 730.407,Z 1231.661,A -85,B 0,C 180,E1 2065.836,E2 2065.836} C_VEL
LIN {X 0,Y 730.461,Z 1235.17,A -85,B 0,C 180,E1 2068.811,E2 2068.811} C_VEL
LIN {X 0,Y 730.52,Z 1234.221,A -85,B 0,C 180,E1 2072.377,E2 2072.377} C_VEL
LIN {X 0,Y 730.507,Z 1227.634,A -85,B 0,C 180,E1 2075.953,E2 2075.953} C_VEL
LIN {X 0,Y 730.509,Z 1216.52,A -85,B 0,C 180,E1 2079.251,E2 2079.251} C_VEL
LIN {X 0,Y 730.623,Z 1198.998,A -85,B 0,C 180,E1 2082.714,E2 2082.714} C_VEL
LIN {X 0,Y 730.868,Z 1176.758,A -85,B 0,C 180,E1 2085.945,E2 2085.945} C_VEL
LIN {X 0,Y 731.326,Z 1149.08,A -85,B 0,C 180,E1 2089.046,E2 2089.046} C_VEL
LIN {X 0,Y 731.961,Z 1116.878,A -85,B 0,C 180,E1 2091.878,E2 2091.878} C_VEL
LIN {X 0,Y 732.766,Z 1079.946,A -85,B 0,C 180,E1 2094.43,E2 2094.43} C_VEL
LIN {X 0,Y 733.605,Z 1038.619,A -85,B 0,C 180,E1 2096.626,E2 2096.626} C_VEL
LIN {X 0,Y 734.388,Z 996.341,A -85,B 0,C 180,E1 2098.293,E2 2098.293} C_VEL
LIN {X 0,Y 734.993,Z 954.775,A -85,B 0,C 180,E1 2099.448,E2 2099.448} C_VEL
LIN {X 0,Y 735.261,Z 911.354,A -85,B 0,C 180,E1 2100.189,E2 2100.189} C_VEL
LIN {X 0,Y 734.609,Z 871.239,A -85,B 0,C 180,E1 2100.671,E2 2100.671} C_VEL
LIN {X 0,Y 730.313,Z 859.31,A -85,B 0,C 180,E1 2101.07,E2 2101.07} C_VEL
LIN {X 0,Y 730.032,Z 859.31,A -85,B 0,C 180,E1 2105.971,E2 2105.971} C_VEL
LIN {X 0,Y 729.879,Z 859.31,A -85,B 0,C 180,E1 2110.06,E2 2110.06} C_VEL
LIN {X 0,Y 730.153,Z 859.31,A -85,B 0,C 180,E1 2115.134,E2 2115.134} C_VEL
LIN {X 0,Y 730.047,Z 859.31,A -85,B 0,C 180,E1 2120.172,E2 2120.172} C_VEL
LIN {X 0,Y 729.991,Z 859.31,A -85,B 0,C 180,E1 2125.921,E2 2125.921} C_VEL
LIN {X 0,Y 730.001,Z 859.31,A -85,B 0,C 180,E1 2130.67,E2 2130.67} C_VEL
LIN {X 0,Y 730.193,Z 859.31,A -85,B 0,C 180,E1 2134.17,E2 2134.17} C_VEL
LIN {X 0,Y 730.085,Z 859.31,A -85,B 0,C 180,E1 2139.063,E2 2139.063} C_VEL
LIN {X 0,Y 730.181,Z 859.31,A -85,B 0,C 180,E1 2143.113,E2 2143.113} C_VEL
LIN {X 0,Y 729.997,Z 859.31,A -85,B 0,C 180,E1 2148.021,E2 2148.021} C_VEL
LIN {X 0,Y 730.312,Z 859.31,A -85,B 0,C 180,E1 2152.849,E2 2152.849} C_VEL
LIN {X 0,Y 730.364,Z 859.31,A -85,B 0,C 180,E1 2157.621,E2 2157.621} C_VEL
LIN {X 0,Y 730.214,Z 859.31,A -85,B 0,C 180,E1 2162.376,E2 2162.376} C_VEL
LIN {X 0,Y 730.192,Z 859.31,A -85,B 0,C 180,E1 2165.952,E2 2165.952} C_VEL
LIN {X 0,Y 730.127,Z 859.31,A -85,B 0,C 180,E1 2170.761,E2 2170.761} C_VEL
LIN {X 0,Y 730.212,Z 859.31,A -85,B 0,C 180,E1 2175.645,E2 2175.645} C_VEL
LIN {X 0,Y 730.108,Z 859.31,A -85,B 0,C 180,E1 2180.942,E2 2180.942} C_VEL
LIN {X 0,Y 730.001,Z 859.31,A -85,B 0,C 180,E1 2185.834,E2 2185.834} C_VEL
LIN {X 0,Y 729.991,Z 859.31,A -85,B 0,C 180,E1 2189.869,E2 2189.869} C_VEL
LIN {X 0,Y 729.968,Z 859.31,A -85,B 0,C 180,E1 2194.076,E2 2194.076} C_VEL
LIN {X 0,Y 729.973,Z 859.31,A -85,B 0,C 180,E1 2198.503,E2 2198.503} C_VEL
LIN {X 0,Y 729.916,Z 859.31,A -85,B 0,C 180,E1 2203.399,E2 2203.399} C_VEL
LIN {X 0,Y 729.962,Z 859.31,A -85,B 0,C 180,E1 2208.374,E2 2208.374} C_VEL
LIN {X 0,Y 730.155,Z 859.31,A -85,B 0,C 180,E1 2212.999,E2 2212.999} C_VEL
LIN {X 0,Y 730.048,Z 859.31,A -85,B 0,C 180,E1 2217.34,E2 2217.34} C_VEL
LIN {X 0,Y 730.021,Z 859.31,A -85,B 0,C 180,E1 2222.829,E2 2222.829} C_VEL
LIN {X 0,Y 730.196,Z 859.31,A -85,B 0,C 180,E1 2225.274,E2 2225.274} C_VEL
LIN {X 0,Y 733.543,Z 872.563,A -85,B 0,C 180,E1 2225.54,E2 2225.54} C_VEL
LIN {X 0,Y 733.467,Z 968.944,A -85,B 0,C 180,E1 2226.637,E2 2226.637} C_VEL
LIN {X 0,Y 733.052,Z 1008.972,A -85,B 0,C 180,E1 2227.575,E2 2227.575} C_VEL
LIN {X 0,Y 732.509,Z 1047.985,A -85,B 0,C 180,E1 2229.006,E2 2229.006} C_VEL
LIN {X 0,Y 731.915,Z 1084.332,A -85,B 0,C 180,E1 2230.891,E2 2230.891} C_VEL
LIN {X 0,Y 731.412,Z 1116.623,A -85,B 0,C 180,E1 2233.14,E2 2233.14} C_VEL
LIN {X 0,Y 730.97,Z 1143.549,A -85,B 0,C 180,E1 2235.596,E2 2235.596} C_VEL
LIN {X 0,Y 730.742,Z 1166.32,A -85,B 0,C 180,E1 2238.336,E2 2238.336} C_VEL
LIN {X 0,Y 730.526,Z 1183.02,A -85,B 0,C 180,E1 2241.05,E2 2241.05} C_VEL
LIN {X 0,Y 730.473,Z 1195.748,A -85,B 0,C 180,E1 2244.047,E2 2244.047} C_VEL
LIN {X 0,Y 730.435,Z 1202.019,A -85,B 0,C 180,E1 2246.432,E2 2246.432} C_VEL
LIN {X 0,Y 730.39,Z 1205.12,A -85,B 0,C 180,E1 2248.811,E2 2248.811} C_VEL
LIN {X 0,Y 730.436,Z 1205.043,A -85,B 0,C 180,E1 2251.189,E2 2251.189} C_VEL
LIN {X 0,Y 730.508,Z 1200.607,A -85,B 0,C 180,E1 2254.164,E2 2254.164} C_VEL
LIN {X 0,Y 730.584,Z 1189.725,A -85,B 0,C 180,E1 2257.448,E2 2257.448} C_VEL
LIN {X 0,Y 730.664,Z 1173.704,A -85,B 0,C 180,E1 2260.48,E2 2260.48} C_VEL
LIN {X 0,Y 730.916,Z 1152.458,A -85,B 0,C 180,E1 2263.335,E2 2263.335} C_VEL
LIN {X 0,Y 731.28,Z 1126.578,A -85,B 0,C 180,E1 2265.936,E2 2265.936} C_VEL
LIN {X 0,Y 731.713,Z 1096.361,A -85,B 0,C 180,E1 2268.254,E2 2268.254} C_VEL
LIN {X 0,Y 732.254,Z 1062.9,A -85,B 0,C 180,E1 2270.199,E2 2270.199} C_VEL
LIN {X 0,Y 732.787,Z 1025.709,A -85,B 0,C 180,E1 2271.788,E2 2271.788} C_VEL
LIN {X 0,Y 733.299,Z 984.8,A -85,B 0,C 180,E1 2272.965,E2 2272.965} C_VEL
LIN {X 0,Y 733.525,Z 943.423,A -85,B 0,C 180,E1 2273.626,E2 2273.626} C_VEL
LIN {X 0,Y 732.914,Z 867.797,A -85,B 0,C 180,E1 2274.442,E2 2274.442} C_VEL
LIN {X 0,Y 730.074,Z 859.31,A -85,B 0,C 180,E1 2274.656,E2 2274.656} C_VEL
LIN {X 0,Y 730.004,Z 859.31,A -85,B 0,C 180,E1 2279.88,E2 2279.88} C_VEL
LIN {X 0,Y 729.991,Z 859.31,A -85,B 0,C 180,E1 2284.088,E2 2284.088} C_VEL
LIN {X 0,Y 730.006,Z 859.31,A -85,B 0,C 180,E1 2288.515,E2 2288.515} C_VEL
LIN {X 0,Y 729.882,Z 859.31,A -85,B 0,C 180,E1 2293.414,E2 2293.414} C_VEL
LIN {X 0,Y 729.937,Z 859.31,A -85,B 0,C 180,E1 2298.387,E2 2298.387} C_VEL
LIN {X 0,Y 730.143,Z 859.31,A -85,B 0,C 180,E1 2303.011,E2 2303.011} C_VEL
LIN {X 0,Y 730.036,Z 859.31,A -85,B 0,C 180,E1 2307.351,E2 2307.351} C_VEL
LIN {X 0,Y 730.071,Z 859.31,A -85,B 0,C 180,E1 2312.841,E2 2312.841} C_VEL
LIN {X 0,Y 730.142,Z 859.31,A -85,B 0,C 180,E1 2316.785,E2 2316.785} C_VEL
LIN {X 0,Y 730.041,Z 859.31,A -85,B 0,C 180,E1 2320.611,E2 2320.611} C_VEL
LIN {X 0,Y 730.084,Z 859.31,A -85,B 0,C 180,E1 2325.584,E2 2325.584} C_VEL
LIN {X 0,Y 730.255,Z 859.31,A -85,B 0,C 180,E1 2330.449,E2 2330.449} C_VEL
LIN {X 0,Y 730.185,Z 859.31,A -85,B 0,C 180,E1 2335.241,E2 2335.241} C_VEL
LIN {X 0,Y 730.298,Z 859.31,A -85,B 0,C 180,E1 2340.002,E2 2340.002} C_VEL
LIN {X 0,Y 730.354,Z 859.31,A -85,B 0,C 180,E1 2345.117,E2 2345.117} C_VEL
LIN {X 0,Y 726.206,Z 859.31,A -85,B 0,C 180,E1 2346.451,E2 2346.451} C_VEL
LIN {X 0,Y 722.282,Z 859.31,A -85,B 0,C 180,E1 2347.8,E2 2347.8} C_VEL
LIN {X 0,Y 722.257,Z 859.31,A -85,B 0,C 180,E1 2353.341,E2 2353.341} C_VEL
LIN {X 0,Y 722.241,Z 859.31,A -85,B 0,C 180,E1 2358.34,E2 2358.34} C_VEL
LIN {X 0,Y 722.26,Z 859.31,A -85,B 0,C 180,E1 2363.487,E2 2363.487} C_VEL
LIN {X 0,Y 722.151,Z 859.31,A -85,B 0,C 180,E1 2368.849,E2 2368.849} C_VEL
LIN {X 0,Y 722.141,Z 859.31,A -85,B 0,C 180,E1 2373.055,E2 2373.055} C_VEL
LIN {X 0,Y 722.144,Z 859.31,A -85,B 0,C 180,E1 2377.473,E2 2377.473} C_VEL
LIN {X 0,Y 721.99,Z 859.31,A -85,B 0,C 180,E1 2382.729,E2 2382.729} C_VEL
LIN {X 0,Y 721.974,Z 859.31,A -85,B 0,C 180,E1 2387.807,E2 2387.807} C_VEL
LIN {X 0,Y 722.273,Z 859.31,A -85,B 0,C 180,E1 2392.848,E2 2392.848} C_VEL
LIN {X 0,Y 722.323,Z 859.31,A -85,B 0,C 180,E1 2398.597,E2 2398.597} C_VEL
LIN {X 0,Y 728.448,Z 875.853,A -85,B 0,C 180,E1 2399.093,E2 2399.093} C_VEL
LIN {X 0,Y 728.205,Z 940.147,A -85,B 0,C 180,E1 2399.936,E2 2399.936} C_VEL
LIN {X 0,Y 727.363,Z 984.393,A -85,B 0,C 180,E1 2401.018,E2 2401.018} C_VEL
LIN {X 0,Y 726.553,Z 1027.042,A -85,B 0,C 180,E1 2402.572,E2 2402.572} C_VEL
LIN {X 0,Y 725.625,Z 1067.507,A -85,B 0,C 180,E1 2404.57,E2 2404.57} C_VEL
LIN {X 0,Y 724.647,Z 1106.819,A -85,B 0,C 180,E1 2407.112,E2 2407.112} C_VEL
LIN {X 0,Y 723.847,Z 1140.994,A -85,B 0,C 180,E1 2409.953,E2 2409.953} C_VEL
LIN {X 0,Y 723.163,Z 1170.555,A -85,B 0,C 180,E1 2413.098,E2 2413.098} C_VEL
LIN {X 0,Y 722.822,Z 1192.207,A -85,B 0,C 180,E1 2416.049,E2 2416.049} C_VEL
LIN {X 0,Y 722.67,Z 1211.082,A -85,B 0,C 180,E1 2419.416,E2 2419.416} C_VEL
LIN {X 0,Y 722.526,Z 1224.158,A -85,B 0,C 180,E1 2422.771,E2 2422.771} C_VEL
LIN {X 0,Y 722.538,Z 1231.662,A -85,B 0,C 180,E1 2425.79,E2 2425.79} C_VEL
LIN {X 0,Y 722.589,Z 1235.17,A -85,B 0,C 180,E1 2428.798,E2 2428.798} C_VEL
LIN {X 0,Y 722.633,Z 1234.22,A -85,B 0,C 180,E1 2432.403,E2 2432.403} C_VEL
LIN {X 0,Y 722.594,Z 1227.634,A -85,B 0,C 180,E1 2436.018,E2 2436.018} C_VEL
LIN {X 0,Y 722.648,Z 1216.52,A -85,B 0,C 180,E1 2439.352,E2 2439.352} C_VEL
LIN {X 0,Y 722.801,Z 1198.195,A -85,B 0,C 180,E1 2442.995,E2 2442.995} C_VEL
LIN {X 0,Y 723.09,Z 1175.544,A -85,B 0,C 180,E1 2446.277,E2 2446.277} C_VEL
LIN {X 0,Y 723.611,Z 1149.079,A -85,B 0,C 180,E1 2449.257,E2 2449.257} C_VEL
LIN {X 0,Y 724.411,Z 1116.879,A -85,B 0,C 180,E1 2452.118,E2 2452.118} C_VEL
LIN {X 0,Y 725.375,Z 1079.948,A -85,B 0,C 180,E1 2454.695,E2 2454.695} C_VEL
LIN {X 0,Y 726.405,Z 1038.624,A -85,B 0,C 180,E1 2456.911,E2 2456.911} C_VEL
LIN {X 0,Y 727.328,Z 996.912,A -85,B 0,C 180,E1 2458.573,E2 2458.573} C_VEL
LIN {X 0,Y 728.086,Z 956.466,A -85,B 0,C 180,E1 2459.719,E2 2459.719} C_VEL
LIN {X 0,Y 728.429,Z 911.969,A -85,B 0,C 180,E1 2460.494,E2 2460.494} C_VEL
LIN {X 0,Y 728.011,Z 873.687,A -85,B 0,C 180,E1 2460.952,E2 2460.952} C_VEL
LIN {X 0,Y 722.386,Z 859.31,A -85,B 0,C 180,E1 2461.402,E2 2461.402} C_VEL
LIN {X 0,Y 722.21,Z 859.31,A -85,B 0,C 180,E1 2467.478,E2 2467.478} C_VEL
LIN {X 0,Y 722.192,Z 859.31,A -85,B 0,C 180,E1 2472.761,E2 2472.761} C_VEL
LIN {X 0,Y 721.954,Z 859.31,A -85,B 0,C 180,E1 2477.274,E2 2477.274} C_VEL
LIN {X 0,Y 722.009,Z 859.31,A -85,B 0,C 180,E1 2482.519,E2 2482.519} C_VEL
LIN {X 0,Y 722.063,Z 859.31,A -85,B 0,C 180,E1 2487.079,E2 2487.079} C_VEL
LIN {X 0,Y 722.097,Z 859.31,A -85,B 0,C 180,E1 2491.806,E2 2491.806} C_VEL
LIN {X 0,Y 722.275,Z 859.31,A -85,B 0,C 180,E1 2496.514,E2 2496.514} C_VEL
LIN {X 0,Y 722.254,Z 859.31,A -85,B 0,C 180,E1 2501.661,E2 2501.661} C_VEL
LIN {X 0,Y 722.111,Z 859.31,A -85,B 0,C 180,E1 2506.656,E2 2506.656} C_VEL
LIN {X 0,Y 722.322,Z 859.31,A -85,B 0,C 180,E1 2510.39,E2 2510.39} C_VEL
LIN {X 0,Y 722.298,Z 859.31,A -85,B 0,C 180,E1 2515.186,E2 2515.186} C_VEL
LIN {X 0,Y 722.382,Z 859.31,A -85,B 0,C 180,E1 2519.998,E2 2519.998} C_VEL
LIN {X 0,Y 722.564,Z 859.31,A -85,B 0,C 180,E1 2524.809,E2 2524.809} C_VEL
LIN {X 0,Y 722.267,Z 859.31,A -85,B 0,C 180,E1 2529.658,E2 2529.658} C_VEL
LIN {X 0,Y 722.175,Z 859.31,A -85,B 0,C 180,E1 2534.578,E2 2534.578} C_VEL
LIN {X 0,Y 722.267,Z 859.31,A -85,B 0,C 180,E1 2539.606,E2 2539.606} C_VEL
LIN {X 0,Y 722.179,Z 859.31,A -85,B 0,C 180,E1 2544.803,E2 2544.803} C_VEL
LIN {X 0,Y 722.059,Z 859.31,A -85,B 0,C 180,E1 2550.231,E2 2550.231} C_VEL
LIN {X 0,Y 722.036,Z 859.31,A -85,B 0,C 180,E1 2555.068,E2 2555.068} C_VEL
LIN {X 0,Y 721.972,Z 859.31,A -85,B 0,C 180,E1 2559.053,E2 2559.053} C_VEL
LIN {X 0,Y 721.946,Z 859.31,A -85,B 0,C 180,E1 2563.822,E2 2563.822} C_VEL
LIN {X 0,Y 721.966,Z 859.31,A -85,B 0,C 180,E1 2569.056,E2 2569.056} C_VEL
LIN {X 0,Y 722.212,Z 859.31,A -85,B 0,C 180,E1 2574.022,E2 2574.022} C_VEL
LIN {X 0,Y 722.066,Z 859.31,A -85,B 0,C 180,E1 2578.356,E2 2578.356} C_VEL
LIN {X 0,Y 722.088,Z 859.31,A -85,B 0,C 180,E1 2582.505,E2 2582.505} C_VEL
LIN {X 0,Y 722.251,Z 859.31,A -85,B 0,C 180,E1 2584.973,E2 2584.973} C_VEL
LIN {X 0,Y 726.416,Z 874.143,A -85,B 0,C 180,E1 2585.302,E2 2585.302} C_VEL
LIN {X 0,Y 726.209,Z 967.455,A -85,B 0,C 180,E1 2586.365,E2 2586.365} C_VEL
LIN {X 0,Y 725.746,Z 1007.033,A -85,B 0,C 180,E1 2587.281,E2 2587.281} C_VEL
LIN {X 0,Y 725.1,Z 1045.199,A -85,B 0,C 180,E1 2588.661,E2 2588.661} C_VEL
LIN {X 0,Y 724.391,Z 1081.767,A -85,B 0,C 180,E1 2590.526,E2 2590.526} C_VEL
LIN {X 0,Y 723.711,Z 1114.318,A -85,B 0,C 180,E1 2592.767,E2 2592.767} C_VEL
LIN {X 0,Y 723.18,Z 1142.357,A -85,B 0,C 180,E1 2595.312,E2 2595.312} C_VEL
LIN {X 0,Y 722.883,Z 1165.224,A -85,B 0,C 180,E1 2598.054,E2 2598.054} C_VEL
LIN {X 0,Y 722.652,Z 1183.018,A -85,B 0,C 180,E1 2600.952,E2 2600.952} C_VEL
LIN {X 0,Y 722.572,Z 1195.747,A -85,B 0,C 180,E1 2603.981,E2 2603.981} C_VEL
LIN {X 0,Y 722.539,Z 1202.018,A -85,B 0,C 180,E1 2606.393,E2 2606.393} C_VEL
LIN {X 0,Y 722.491,Z 1205.12,A -85,B 0,C 180,E1 2608.798,E2 2608.798} C_VEL
LIN {X 0,Y 722.565,Z 1205.043,A -85,B 0,C 180,E1 2611.202,E2 2611.202} C_VEL
LIN {X 0,Y 722.626,Z 1200.609,A -85,B 0,C 180,E1 2614.209,E2 2614.209} C_VEL
LIN {X 0,Y 722.701,Z 1189.728,A -85,B 0,C 180,E1 2617.53,E2 2617.53} C_VEL
LIN {X 0,Y 722.8,Z 1173.671,A -85,B 0,C 180,E1 2620.601,E2 2620.601} C_VEL
LIN {X 0,Y 723.102,Z 1152.464,A -85,B 0,C 180,E1 2623.482,E2 2623.482} C_VEL
LIN {X 0,Y 723.54,Z 1126.584,A -85,B 0,C 180,E1 2626.111,E2 2626.111} C_VEL
LIN {X 0,Y 724.064,Z 1096.367,A -85,B 0,C 180,E1 2628.453,E2 2628.453} C_VEL
LIN {X 0,Y 724.741,Z 1062.268,A -85,B 0,C 180,E1 2630.451,E2 2630.451} C_VEL
LIN {X 0,Y 725.45,Z 1023.989,A -85,B 0,C 180,E1 2632.085,E2 2632.085} C_VEL
LIN {X 0,Y 726.039,Z 983.605,A -85,B 0,C 180,E1 2633.234,E2 2633.234} C_VEL
LIN {X 0,Y 726.282,Z 941.818,A -85,B 0,C 180,E1 2633.894,E2 2633.894} C_VEL
LIN {X 0,Y 725.562,Z 869.487,A -85,B 0,C 180,E1 2634.689,E2 2634.689} C_VEL
LIN {X 0,Y 722.13,Z 859.31,A -85,B 0,C 180,E1 2634.953,E2 2634.953} C_VEL
LIN {X 0,Y 722.069,Z 859.31,A -85,B 0,C 180,E1 2640.242,E2 2640.242} C_VEL
LIN {X 0,Y 722.048,Z 859.31,A -85,B 0,C 180,E1 2645.094,E2 2645.094} C_VEL
LIN {X 0,Y 722.014,Z 859.31,A -85,B 0,C 180,E1 2649.078,E2 2649.078} C_VEL
LIN {X 0,Y 721.912,Z 859.31,A -85,B 0,C 180,E1 2653.842,E2 2653.842} C_VEL
LIN {X 0,Y 721.95,Z 859.31,A -85,B 0,C 180,E1 2659.078,E2 2659.078} C_VEL
LIN {X 0,Y 722.202,Z 859.31,A -85,B 0,C 180,E1 2664.034,E2 2664.034} C_VEL
LIN {X 0,Y 722.018,Z 859.31,A -85,B 0,C 180,E1 2668.365,E2 2668.365} C_VEL
LIN {X 0,Y 722.133,Z 859.31,A -85,B 0,C 180,E1 2672.517,E2 2672.517} C_VEL
LIN {X 0,Y 722.175,Z 859.31,A -85,B 0,C 180,E1 2677.402,E2 2677.402} C_VEL
LIN {X 0,Y 721.907,Z 859.31,A -85,B 0,C 180,E1 2681.655,E2 2681.655} C_VEL
LIN {X 0,Y 722.114,Z 859.31,A -85,B 0,C 180,E1 2686.66,E2 2686.66} C_VEL
LIN {X 0,Y 722.366,Z 859.31,A -85,B 0,C 180,E1 2690.371,E2 2690.371} C_VEL
LIN {X 0,Y 722.306,Z 859.31,A -85,B 0,C 180,E1 2695.189,E2 2695.189} C_VEL
LIN {X 0,Y 722.406,Z 859.31,A -85,B 0,C 180,E1 2700.002,E2 2700.002} C_VEL
LIN {X 0,Y 722.454,Z 859.31,A -85,B 0,C 180,E1 2705.103,E2 2705.103} C_VEL
LIN {X 0,Y 722.282,Z 859.31,A -85,B 0,C 180,E1 2707.8,E2 2707.8} C_VEL
LIN {X 0,Y 719.784,Z 859.31,A -85,B 0,C 180,E1 2708.821,E2 2708.821} C_VEL
LIN {X 0,Y 714.37,Z 859.31,A -85,B 0,C 180,E1 2710.344,E2 2710.344} C_VEL
LIN {X 0,Y 714.274,Z 859.31,A -85,B 0,C 180,E1 2710.521,E2 2710.521} C_VEL
LIN {X 0,Y 714.289,Z 859.31,A -85,B 0,C 180,E1 2714.746,E2 2714.746} C_VEL
LIN {X 0,Y 714.393,Z 859.31,A -85,B 0,C 180,E1 2719.835,E2 2719.835} C_VEL
LIN {X 0,Y 714.287,Z 859.31,A -85,B 0,C 180,E1 2725.1,E2 2725.1} C_VEL
LIN {X 0,Y 714.162,Z 859.31,A -85,B 0,C 180,E1 2729.549,E2 2729.549} C_VEL
LIN {X 0,Y 714.125,Z 859.31,A -85,B 0,C 180,E1 2734.153,E2 2734.153} C_VEL
LIN {X 0,Y 714.107,Z 859.31,A -85,B 0,C 180,E1 2738.268,E2 2738.268} C_VEL
LIN {X 0,Y 714.044,Z 859.31,A -85,B 0,C 180,E1 2743.819,E2 2743.819} C_VEL
LIN {X 0,Y 714.013,Z 859.31,A -85,B 0,C 180,E1 2748.861,E2 2748.861} C_VEL
LIN {X 0,Y 714.332,Z 859.31,A -85,B 0,C 180,E1 2753.697,E2 2753.697} C_VEL
LIN {X 0,Y 714.392,Z 859.31,A -85,B 0,C 180,E1 2758.217,E2 2758.217} C_VEL
LIN {X 0,Y 721.708,Z 877.996,A -85,B 0,C 180,E1 2758.797,E2 2758.797} C_VEL
LIN {X 0,Y 721.329,Z 941.543,A -85,B 0,C 180,E1 2759.645,E2 2759.645} C_VEL
LIN {X 0,Y 720.378,Z 987.233,A -85,B 0,C 180,E1 2760.797,E2 2760.797} C_VEL
LIN {X 0,Y 719.353,Z 1029.651,A -85,B 0,C 180,E1 2762.392,E2 2762.392} C_VEL
LIN {X 0,Y 718.264,Z 1068.895,A -85,B 0,C 180,E1 2764.375,E2 2764.375} C_VEL
LIN {X 0,Y 717.164,Z 1107.038,A -85,B 0,C 180,E1 2766.877,E2 2766.877} C_VEL
LIN {X 0,Y 716.236,Z 1140.985,A -85,B 0,C 180,E1 2769.73,E2 2769.73} C_VEL
LIN {X 0,Y 715.415,Z 1170.553,A -85,B 0,C 180,E1 2772.909,E2 2772.909} C_VEL
LIN {X 0,Y 714.95,Z 1194.178,A -85,B 0,C 180,E1 2776.206,E2 2776.206} C_VEL
LIN {X 0,Y 714.804,Z 1211.137,A -85,B 0,C 180,E1 2779.31,E2 2779.31} C_VEL
LIN {X 0,Y 714.667,Z 1224.158,A -85,B 0,C 180,E1 2782.691,E2 2782.691} C_VEL
LIN {X 0,Y 714.641,Z 1231.662,A -85,B 0,C 180,E1 2785.744,E2 2785.744} C_VEL
LIN {X 0,Y 714.687,Z 1235.169,A -85,B 0,C 180,E1 2788.785,E2 2788.785} C_VEL
LIN {X 0,Y 714.726,Z 1234.22,A -85,B 0,C 180,E1 2792.43,E2 2792.43} C_VEL
LIN {X 0,Y 714.696,Z 1227.635,A -85,B 0,C 180,E1 2796.085,E2 2796.085} C_VEL
LIN {X 0,Y 714.778,Z 1216.519,A -85,B 0,C 180,E1 2799.456,E2 2799.456} C_VEL
LIN {X 0,Y 714.922,Z 1198.219,A -85,B 0,C 180,E1 2803.137,E2 2803.137} C_VEL
LIN {X 0,Y 715.286,Z 1175.546,A -85,B 0,C 180,E1 2806.46,E2 2806.46} C_VEL
LIN {X 0,Y 715.922,Z 1149.644,A -85,B 0,C 180,E1 2809.416,E2 2809.416} C_VEL
LIN {X 0,Y 716.876,Z 1116.88,A -85,B 0,C 180,E1 2812.363,E2 2812.363} C_VEL
LIN {X 0,Y 718.014,Z 1079.949,A -85,B 0,C 180,E1 2814.966,E2 2814.966} C_VEL
LIN {X 0,Y 719.193,Z 1038.879,A -85,B 0,C 180,E1 2817.19,E2 2817.19} C_VEL
LIN {X 0,Y 720.281,Z 997.561,A -85,B 0,C 180,E1 2818.855,E2 2818.855} C_VEL
LIN {X 0,Y 721.174,Z 956.501,A -85,B 0,C 180,E1 2820.032,E2 2820.032} C_VEL
LIN {X 0,Y 721.614,Z 913.562,A -85,B 0,C 180,E1 2820.792,E2 2820.792} C_VEL
LIN {X 0,Y 721.254,Z 875.632,A -85,B 0,C 180,E1 2821.252,E2 2821.252} C_VEL
LIN {X 0,Y 714.447,Z 859.31,A -85,B 0,C 180,E1 2821.811,E2 2821.811} C_VEL
LIN {X 0,Y 714.249,Z 859.31,A -85,B 0,C 180,E1 2826.443,E2 2826.443} C_VEL
LIN {X 0,Y 714.205,Z 859.31,A -85,B 0,C 180,E1 2832.063,E2 2832.063} C_VEL
LIN {X 0,Y 714.174,Z 859.31,A -85,B 0,C 180,E1 2836.169,E2 2836.169} C_VEL
LIN {X 0,Y 714.083,Z 859.31,A -85,B 0,C 180,E1 2841.734,E2 2841.734} C_VEL
LIN {X 0,Y 714.101,Z 859.31,A -85,B 0,C 180,E1 2846.524,E2 2846.524} C_VEL
LIN {X 0,Y 714.151,Z 859.31,A -85,B 0,C 180,E1 2850.796,E2 2850.796} C_VEL
LIN {X 0,Y 714.296,Z 859.31,A -85,B 0,C 180,E1 2855.81,E2 2855.81} C_VEL
LIN {X 0,Y 714.266,Z 859.31,A -85,B 0,C 180,E1 2860.161,E2 2860.161} C_VEL
LIN {X 0,Y 714.296,Z 859.31,A -85,B 0,C 180,E1 2865.254,E2 2865.254} C_VEL
LIN {X 0,Y 714.422,Z 859.31,A -85,B 0,C 180,E1 2870.232,E2 2870.232} C_VEL
LIN {X 0,Y 714.422,Z 859.31,A -85,B 0,C 180,E1 2875.465,E2 2875.465} C_VEL
LIN {X 0,Y 714.482,Z 859.31,A -85,B 0,C 180,E1 2879.998,E2 2879.998} C_VEL
LIN {X 0,Y 714.666,Z 859.31,A -85,B 0,C 180,E1 2884.862,E2 2884.862} C_VEL
LIN {X 0,Y 714.351,Z 859.31,A -85,B 0,C 180,E1 2889.766,E2 2889.766} C_VEL
LIN {X 0,Y 714.293,Z 859.31,A -85,B 0,C 180,E1 2894.742,E2 2894.742} C_VEL
LIN {X 0,Y 714.337,Z 859.31,A -85,B 0,C 180,E1 2899.833,E2 2899.833} C_VEL
LIN {X 0,Y 714.25,Z 859.31,A -85,B 0,C 180,E1 2905.098,E2 2905.098} C_VEL
LIN {X 0,Y 714.138,Z 859.31,A -85,B 0,C 180,E1 2909.547,E2 2909.547} C_VEL
LIN {X 0,Y 714.121,Z 859.31,A -85,B 0,C 180,E1 2914.153,E2 2914.153} C_VEL
LIN {X 0,Y 714.125,Z 859.31,A -85,B 0,C 180,E1 2918.27,E2 2918.27} C_VEL
LIN {X 0,Y 714.047,Z 859.31,A -85,B 0,C 180,E1 2923.82,E2 2923.82} C_VEL
LIN {X 0,Y 714.052,Z 859.31,A -85,B 0,C 180,E1 2928.864,E2 2928.864} C_VEL
LIN {X 0,Y 714.296,Z 859.31,A -85,B 0,C 180,E1 2933.695,E2 2933.695} C_VEL
LIN {X 0,Y 714.173,Z 859.31,A -85,B 0,C 180,E1 2938.043,E2 2938.043} C_VEL
LIN {X 0,Y 714.137,Z 859.31,A -85,B 0,C 180,E1 2942.988,E2 2942.988} C_VEL
LIN {X 0,Y 714.295,Z 859.31,A -85,B 0,C 180,E1 2944.691,E2 2944.691} C_VEL
LIN {X 0,Y 719.256,Z 875.787,A -85,B 0,C 180,E1 2945.057,E2 2945.057} C_VEL
LIN {X 0,Y 718.966,Z 968.269,A -85,B 0,C 180,E1 2946.126,E2 2946.126} C_VEL
LIN {X 0,Y 718.406,Z 1007.887,A -85,B 0,C 180,E1 2947.061,E2 2947.061} C_VEL
LIN {X 0,Y 717.631,Z 1046.51,A -85,B 0,C 180,E1 2948.485,E2 2948.485} C_VEL
LIN {X 0,Y 716.784,Z 1083.04,A -85,B 0,C 180,E1 2950.391,E2 2950.391} C_VEL
LIN {X 0,Y 716.013,Z 1114.731,A -85,B 0,C 180,E1 2952.611,E2 2952.611} C_VEL
LIN {X 0,Y 715.417,Z 1142.491,A -85,B 0,C 180,E1 2955.164,E2 2955.164} C_VEL
LIN {X 0,Y 715.052,Z 1165.222,A -85,B 0,C 180,E1 2957.921,E2 2957.921} C_VEL
LIN {X 0,Y 714.771,Z 1183.016,A -85,B 0,C 180,E1 2960.851,E2 2960.851} C_VEL
LIN {X 0,Y 714.678,Z 1195.745,A -85,B 0,C 180,E1 2963.915,E2 2963.915} C_VEL
LIN {X 0,Y 714.641,Z 1202.018,A -85,B 0,C 180,E1 2966.353,E2 2966.353} C_VEL
LIN {X 0,Y 714.591,Z 1205.12,A -85,B 0,C 180,E1 2968.785,E2 2968.785} C_VEL
LIN {X 0,Y 714.664,Z 1205.044,A -85,B 0,C 180,E1 2971.215,E2 2971.215} C_VEL
LIN {X 0,Y 714.741,Z 1200.61,A -85,B 0,C 180,E1 2974.256,E2 2974.256} C_VEL
LIN {X 0,Y 714.835,Z 1189.73,A -85,B 0,C 180,E1 2977.613,E2 2977.613} C_VEL
LIN {X 0,Y 714.938,Z 1173.872,A -85,B 0,C 180,E1 2980.688,E2 2980.688} C_VEL
LIN {X 0,Y 715.303,Z 1152.467,A -85,B 0,C 180,E1 2983.631,E2 2983.631} C_VEL
LIN {X 0,Y 715.791,Z 1126.59,A -85,B 0,C 180,E1 2986.29,E2 2986.29} C_VEL
LIN {X 0,Y 716.516,Z 1096.372,A -85,B 0,C 180,E1 2988.655,E2 2988.655} C_VEL
LIN {X 0,Y 717.226,Z 1062.866,A -85,B 0,C 180,E1 2990.644,E2 2990.644} C_VEL
LIN {X 0,Y 718.05,Z 1025.161,A -85,B 0,C 180,E1 2992.28,E2 2992.28} C_VEL
LIN {X 0,Y 718.746,Z 985.537,A -85,B 0,C 180,E1 2993.441,E2 2993.441} C_VEL
LIN {X 0,Y 719.081,Z 944.709,A -85,B 0,C 180,E1 2994.118,E2 2994.118} C_VEL
LIN {X 0,Y 718.644,Z 872.137,A -85,B 0,C 180,E1 2994.915,E2 2994.915} C_VEL
LIN {X 0,Y 714.19,Z 859.31,A -85,B 0,C 180,E1 2995.283,E2 2995.283} C_VEL
LIN {X 0,Y 714.187,Z 859.31,A -85,B 0,C 180,E1 3000.611,E2 3000.611} C_VEL
LIN {X 0,Y 714.154,Z 859.31,A -85,B 0,C 180,E1 3004.952,E2 3004.952} C_VEL
LIN {X 0,Y 714.064,Z 859.31,A -85,B 0,C 180,E1 3009.54,E2 3009.54} C_VEL
LIN {X 0,Y 713.983,Z 859.31,A -85,B 0,C 180,E1 3014.456,E2 3014.456} C_VEL
LIN {X 0,Y 714.035,Z 859.31,A -85,B 0,C 180,E1 3018.878,E2 3018.878} C_VEL
LIN {X 0,Y 714.285,Z 859.31,A -85,B 0,C 180,E1 3023.72,E2 3023.72} C_VEL
LIN {X 0,Y 714.132,Z 859.31,A -85,B 0,C 180,E1 3028.076,E2 3028.076} C_VEL
LIN {X 0,Y 714.225,Z 859.31,A -85,B 0,C 180,E1 3033.552,E2 3033.552} C_VEL
LIN {X 0,Y 714.278,Z 859.31,A -85,B 0,C 180,E1 3037.559,E2 3037.559} C_VEL
LIN {X 0,Y 714.07,Z 859.31,A -85,B 0,C 180,E1 3041.446,E2 3041.446} C_VEL
LIN {X 0,Y 714.212,Z 859.31,A -85,B 0,C 180,E1 3046.509,E2 3046.509} C_VEL
LIN {X 0,Y 714.453,Z 859.31,A -85,B 0,C 180,E1 3050.236,E2 3050.236} C_VEL
LIN {X 0,Y 714.416,Z 859.31,A -85,B 0,C 180,E1 3055.136,E2 3055.136} C_VEL
LIN {X 0,Y 714.506,Z 859.31,A -85,B 0,C 180,E1 3060.002,E2 3060.002} C_VEL
LIN {X 0,Y 714.64,Z 859.31,A -85,B 0,C 180,E1 3064.866,E2 3064.866} C_VEL
LIN {X 0,Y 714.35,Z 859.31,A -85,B 0,C 180,E1 3069.769,E2 3069.769} C_VEL
LIN {X 0,Y 714.274,Z 859.31,A -85,B 0,C 180,E1 3070.521,E2 3070.521} C_VEL
LIN {X 0,Y 710.328,Z 859.31,A -85,B 0,C 180,E1 3071.893,E2 3071.893} C_VEL
LIN {X 0,Y 706.39,Z 859.31,A -85,B 0,C 180,E1 3073.281,E2 3073.281} C_VEL
LIN {X 0,Y 706.494,Z 859.31,A -85,B 0,C 180,E1 3077.471,E2 3077.471} C_VEL
LIN {X 0,Y 706.376,Z 859.31,A -85,B 0,C 180,E1 3082.717,E2 3082.717} C_VEL
LIN {X 0,Y 706.297,Z 859.31,A -85,B 0,C 180,E1 3088.157,E2 3088.157} C_VEL
LIN {X 0,Y 706.237,Z 859.31,A -85,B 0,C 180,E1 3093.198,E2 3093.198} C_VEL
LIN {X 0,Y 706.172,Z 859.31,A -85,B 0,C 180,E1 3098.473,E2 3098.473} C_VEL
LIN {X 0,Y 706.164,Z 859.31,A -85,B 0,C 180,E1 3103.354,E2 3103.354} C_VEL
LIN {X 0,Y 706.133,Z 859.31,A -85,B 0,C 180,E1 3108.668,E2 3108.668} C_VEL
LIN {X 0,Y 706.334,Z 859.31,A -85,B 0,C 180,E1 3113.081,E2 3113.081} C_VEL
LIN {X 0,Y 706.49,Z 859.917,A -85,B 0,C 180,E1 3117.834,E2 3117.834} C_VEL
LIN {X 0,Y 714.951,Z 879.825,A -85,B 0,C 180,E1 3118.489,E2 3118.489} C_VEL
LIN {X 0,Y 714.506,Z 941.641,A -85,B 0,C 180,E1 3119.326,E2 3119.326} C_VEL
LIN {X 0,Y 713.38,Z 987.487,A -85,B 0,C 180,E1 3120.491,E2 3120.491} C_VEL
LIN {X 0,Y 712.235,Z 1029.656,A -85,B 0,C 180,E1 3122.092,E2 3122.092} C_VEL
LIN {X 0,Y 710.973,Z 1068.891,A -85,B 0,C 180,E1 3124.093,E2 3124.093} C_VEL
LIN {X 0,Y 709.721,Z 1106.974,A -85,B 0,C 180,E1 3126.615,E2 3126.615} C_VEL
LIN {X 0,Y 708.621,Z 1140.984,A -85,B 0,C 180,E1 3129.503,E2 3129.503} C_VEL
LIN {X 0,Y 707.701,Z 1170.551,A -85,B 0,C 180,E1 3132.717,E2 3132.717} C_VEL
LIN {X 0,Y 707.129,Z 1194.179,A -85,B 0,C 180,E1 3136.05,E2 3136.05} C_VEL
LIN {X 0,Y 706.967,Z 1211.137,A -85,B 0,C 180,E1 3139.19,E2 3139.19} C_VEL
LIN {X 0,Y 706.782,Z 1224.158,A -85,B 0,C 180,E1 3142.609,E2 3142.609} C_VEL
LIN {X 0,Y 706.733,Z 1231.831,A -85,B 0,C 180,E1 3145.782,E2 3145.782} C_VEL
LIN {X 0,Y 706.814,Z 1235.169,A -85,B 0,C 180,E1 3148.771,E2 3148.771} C_VEL
LIN {X 0,Y 706.819,Z 1234.219,A -85,B 0,C 180,E1 3152.457,E2 3152.457} C_VEL
LIN {X 0,Y 706.788,Z 1227.635,A -85,B 0,C 180,E1 3156.154,E2 3156.154} C_VEL
LIN {X 0,Y 706.894,Z 1216.098,A -85,B 0,C 180,E1 3159.66,E2 3159.66} C_VEL
LIN {X 0,Y 707.077,Z 1199.526,A -85,B 0,C 180,E1 3163.05,E2 3163.05} C_VEL
LIN {X 0,Y 707.481,Z 1177.979,A -85,B 0,C 180,E1 3166.326,E2 3166.326} C_VEL
LIN {X 0,Y 708.208,Z 1150.929,A -85,B 0,C 180,E1 3169.505,E2 3169.505} C_VEL
LIN {X 0,Y 709.318,Z 1118.213,A -85,B 0,C 180,E1 3172.509,E2 3172.509} C_VEL
LIN {X 0,Y 710.657,Z 1079.95,A -85,B 0,C 180,E1 3175.242,E2 3175.242} C_VEL
LIN {X 0,Y 712.018,Z 1038.874,A -85,B 0,C 180,E1 3177.487,E2 3177.487} C_VEL
LIN {X 0,Y 713.306,Z 997.653,A -85,B 0,C 180,E1 3179.161,E2 3179.161} C_VEL
LIN {X 0,Y 714.303,Z 956.735,A -85,B 0,C 180,E1 3180.346,E2 3180.346} C_VEL
LIN {X 0,Y 714.86,Z 912.163,A -85,B 0,C 180,E1 3181.134,E2 3181.134} C_VEL
LIN {X 0,Y 714.462,Z 878.024,A -85,B 0,C 180,E1 3181.556,E2 3181.556} C_VEL
LIN {X 0,Y 706.463,Z 859.31,A -85,B 0,C 180,E1 3182.25,E2 3182.25} C_VEL
LIN {X 0,Y 706.255,Z 859.31,A -85,B 0,C 180,E1 3187.471,E2 3187.471} C_VEL
LIN {X 0,Y 706.424,Z 859.31,A -85,B 0,C 180,E1 3193.346,E2 3193.346} C_VEL
LIN {X 0,Y 706.171,Z 859.31,A -85,B 0,C 180,E1 3198.679,E2 3198.679} C_VEL
LIN {X 0,Y 706.13,Z 859.31,A -85,B 0,C 180,E1 3203.078,E2 3203.078} C_VEL
LIN {X 0,Y 706.23,Z 859.31,A -85,B 0,C 180,E1 3207.569,E2 3207.569} C_VEL
LIN {X 0,Y 706.273,Z 859.31,A -85,B 0,C 180,E1 3211.842,E2 3211.842} C_VEL
LIN {X 0,Y 706.404,Z 859.31,A -85,B 0,C 180,E1 3215.953,E2 3215.953} C_VEL
LIN {X 0,Y 706.405,Z 859.31,A -85,B 0,C 180,E1 3221.234,E2 3221.234} C_VEL
LIN {X 0,Y 706.309,Z 859.31,A -85,B 0,C 180,E1 3226.352,E2 3226.352} C_VEL
LIN {X 0,Y 706.399,Z 859.31,A -85,B 0,C 180,E1 3231.365,E2 3231.365} C_VEL
LIN {X 0,Y 706.6,Z 859.31,A -85,B 0,C 180,E1 3236.311,E2 3236.311} C_VEL
LIN {X 0,Y 706.751,Z 859.31,A -85,B 0,C 180,E1 3241.227,E2 3241.227} C_VEL
LIN {X 0,Y 706.472,Z 859.31,A -85,B 0,C 180,E1 3246.153,E2 3246.153} C_VEL
LIN {X 0,Y 706.409,Z 859.31,A -85,B 0,C 180,E1 3251.126,E2 3251.126} C_VEL
LIN {X 0,Y 706.466,Z 859.31,A -85,B 0,C 180,E1 3256.185,E2 3256.185} C_VEL
LIN {X 0,Y 706.361,Z 859.31,A -85,B 0,C 180,E1 3261.38,E2 3261.38} C_VEL
LIN {X 0,Y 706.288,Z 859.31,A -85,B 0,C 180,E1 3265.7,E2 3265.7} C_VEL
LIN {X 0,Y 706.248,Z 859.31,A -85,B 0,C 180,E1 3270.982,E2 3270.982} C_VEL
LIN {X 0,Y 706.246,Z 859.31,A -85,B 0,C 180,E1 3275.388,E2 3275.388} C_VEL
LIN {X 0,Y 706.085,Z 859.31,A -85,B 0,C 180,E1 3280.062,E2 3280.062} C_VEL
LIN {X 0,Y 706.105,Z 859.31,A -85,B 0,C 180,E1 3285.069,E2 3285.069} C_VEL
LIN {X 0,Y 706.093,Z 859.31,A -85,B 0,C 180,E1 3289.924,E2 3289.924} C_VEL
LIN {X 0,Y 706.318,Z 859.31,A -85,B 0,C 180,E1 3294.603,E2 3294.603} C_VEL
LIN {X 0,Y 706.183,Z 859.31,A -85,B 0,C 180,E1 3299.098,E2 3299.098} C_VEL
LIN {X 0,Y 706.351,Z 859.31,A -85,B 0,C 180,E1 3304.369,E2 3304.369} C_VEL
LIN {X 0,Y 712.095,Z 877.858,A -85,B 0,C 180,E1 3304.812,E2 3304.812} C_VEL
LIN {X 0,Y 711.736,Z 968.238,A -85,B 0,C 180,E1 3305.868,E2 3305.868} C_VEL
LIN {X 0,Y 711.096,Z 1008.077,A -85,B 0,C 180,E1 3306.818,E2 3306.818} C_VEL
LIN {X 0,Y 710.187,Z 1047.435,A -85,B 0,C 180,E1 3308.289,E2 3308.289} C_VEL
LIN {X 0,Y 709.214,Z 1084.012,A -85,B 0,C 180,E1 3310.236,E2 3310.236} C_VEL
LIN {X 0,Y 708.328,Z 1115.118,A -85,B 0,C 180,E1 3312.449,E2 3312.449} C_VEL
LIN {X 0,Y 707.681,Z 1141.857,A -85,B 0,C 180,E1 3314.93,E2 3314.93} C_VEL
LIN {X 0,Y 707.222,Z 1165.219,A -85,B 0,C 180,E1 3317.785,E2 3317.785} C_VEL
LIN {X 0,Y 706.913,Z 1183.391,A -85,B 0,C 180,E1 3320.825,E2 3320.825} C_VEL
LIN {X 0,Y 706.781,Z 1195.744,A -85,B 0,C 180,E1 3323.846,E2 3323.846} C_VEL
LIN {X 0,Y 706.774,Z 1202.018,A -85,B 0,C 180,E1 3326.312,E2 3326.312} C_VEL
LIN {X 0,Y 706.705,Z 1205.12,A -85,B 0,C 180,E1 3328.772,E2 3328.772} C_VEL
LIN {X 0,Y 706.792,Z 1205.045,A -85,B 0,C 180,E1 3331.229,E2 3331.229} C_VEL
LIN {X 0,Y 706.839,Z 1200.737,A -85,B 0,C 180,E1 3334.249,E2 3334.249} C_VEL
LIN {X 0,Y 706.903,Z 1191.025,A -85,B 0,C 180,E1 3337.39,E2 3337.39} C_VEL
LIN {X 0,Y 707.067,Z 1175.788,A -85,B 0,C 180,E1 3340.496,E2 3340.496} C_VEL
LIN {X 0,Y 707.483,Z 1153.798,A -85,B 0,C 180,E1 3343.627,E2 3343.627} C_VEL
LIN {X 0,Y 708.029,Z 1128.349,A -85,B 0,C 180,E1 3346.314,E2 3346.314} C_VEL
LIN {X 0,Y 708.784,Z 1098.675,A -85,B 0,C 180,E1 3348.704,E2 3348.704} C_VEL
LIN {X 0,Y 709.7,Z 1064.418,A -85,B 0,C 180,E1 3350.791,E2 3350.791} C_VEL
LIN {X 0,Y 710.629,Z 1027.491,A -85,B 0,C 180,E1 3352.436,E2 3352.436} C_VEL
LIN {X 0,Y 711.409,Z 988.595,A -85,B 0,C 180,E1 3353.621,E2 3353.621} C_VEL
LIN {X 0,Y 711.824,Z 948.736,A -85,B 0,C 180,E1 3354.33,E2 3354.33} C_VEL
LIN {X 0,Y 711.273,Z 873.6,A -85,B 0,C 180,E1 3355.175,E2 3355.175} C_VEL
LIN {X 0,Y 706.238,Z 859.31,A -85,B 0,C 180,E1 3355.582,E2 3355.582} C_VEL
LIN {X 0,Y 706.271,Z 859.31,A -85,B 0,C 180,E1 3360.992,E2 3360.992} C_VEL
LIN {X 0,Y 706.27,Z 859.31,A -85,B 0,C 180,E1 3365.409,E2 3365.409} C_VEL
LIN {X 0,Y 706.132,Z 859.31,A -85,B 0,C 180,E1 3370.074,E2 3370.074} C_VEL
LIN {X 0,Y 706.084,Z 859.31,A -85,B 0,C 180,E1 3375.089,E2 3375.089} C_VEL
LIN {X 0,Y 706.081,Z 859.31,A -85,B 0,C 180,E1 3379.938,E2 3379.938} C_VEL
LIN {X 0,Y 706.337,Z 859.31,A -85,B 0,C 180,E1 3384.617,E2 3384.617} C_VEL
LIN {X 0,Y 706.163,Z 859.31,A -85,B 0,C 180,E1 3389.129,E2 3389.129} C_VEL
LIN {X 0,Y 706.336,Z 859.31,A -85,B 0,C 180,E1 3394.293,E2 3394.293} C_VEL
LIN {X 0,Y 706.395,Z 859.31,A -85,B 0,C 180,E1 3398.621,E2 3398.621} C_VEL
LIN {X 0,Y 706.096,Z 859.31,A -85,B 0,C 180,E1 3403.807,E2 3403.807} C_VEL
LIN {X 0,Y 706.522,Z 859.31,A -85,B 0,C 180,E1 3408.875,E2 3408.875} C_VEL
LIN {X 0,Y 706.631,Z 859.31,A -85,B 0,C 180,E1 3413.848,E2 3413.848} C_VEL
LIN {X 0,Y 706.544,Z 859.31,A -85,B 0,C 180,E1 3418.773,E2 3418.773} C_VEL
LIN {X 0,Y 706.521,Z 859.31,A -85,B 0,C 180,E1 3422.459,E2 3422.459} C_VEL
LIN {X 0,Y 706.475,Z 859.31,A -85,B 0,C 180,E1 3426.156,E2 3426.156} C_VEL
LIN {X 0,Y 706.384,Z 859.31,A -85,B 0,C 180,E1 3431.13,E2 3431.13} C_VEL
LIN {X 0,Y 706.39,Z 859.31,A -85,B 0,C 180,E1 3433.281,E2 3433.281} C_VEL
LIN {X 0,Y 705.131,Z 859.31,A -85,B 0,C 180,E1 3433.985,E2 3433.985} C_VEL
LIN {X 0,Y 698.586,Z 859.31,A -85,B 0,C 180,E1 3435.895,E2 3435.895} C_VEL
LIN {X 0,Y 698.514,Z 859.31,A -85,B 0,C 180,E1 3436.076,E2 3436.076} C_VEL
LIN {X 0,Y 698.524,Z 859.31,A -85,B 0,C 180,E1 3441.126,E2 3441.126} C_VEL
LIN {X 0,Y 698.447,Z 859.31,A -85,B 0,C 180,E1 3445.71,E2 3445.71} C_VEL
LIN {X 0,Y 698.341,Z 859.31,A -85,B 0,C 180,E1 3449.931,E2 3449.931} C_VEL
LIN {X 0,Y 698.272,Z 859.31,A -85,B 0,C 180,E1 3454.449,E2 3454.449} C_VEL
LIN {X 0,Y 698.228,Z 859.31,A -85,B 0,C 180,E1 3458.993,E2 3458.993} C_VEL
LIN {X 0,Y 698.168,Z 859.31,A -85,B 0,C 180,E1 3464.256,E2 3464.256} C_VEL
LIN {X 0,Y 698.163,Z 859.31,A -85,B 0,C 180,E1 3469.417,E2 3469.417} C_VEL
LIN {X 0,Y 698.424,Z 859.31,A -85,B 0,C 180,E1 3474.141,E2 3474.141} C_VEL
LIN {X 0,Y 698.474,Z 859.31,A -85,B 0,C 180,E1 3477.398,E2 3477.398} C_VEL
LIN {X 0,Y 708.188,Z 881.507,A -85,B 0,C 180,E1 3478.173,E2 3478.173} C_VEL
LIN {X 0,Y 707.723,Z 941.38,A -85,B 0,C 180,E1 3478.994,E2 3478.994} C_VEL
LIN {X 0,Y 706.449,Z 986.926,A -85,B 0,C 180,E1 3480.154,E2 3480.154} C_VEL
LIN {X 0,Y 705.137,Z 1029.656,A -85,B 0,C 180,E1 3481.786,E2 3481.786} C_VEL
LIN {X 0,Y 703.63,Z 1070.16,A -85,B 0,C 180,E1 3483.88,E2 3483.88} C_VEL
LIN {X 0,Y 702.241,Z 1106.973,A -85,B 0,C 180,E1 3486.351,E2 3486.351} C_VEL
LIN {X 0,Y 701.011,Z 1140.982,A -85,B 0,C 180,E1 3489.27,E2 3489.27} C_VEL
LIN {X 0,Y 699.928,Z 1171.876,A -85,B 0,C 180,E1 3492.682,E2 3492.682} C_VEL
LIN {X 0,Y 699.268,Z 1196.135,A -85,B 0,C 180,E1 3496.21,E2 3496.21} C_VEL
LIN {X 0,Y 698.998,Z 1213.835,A -85,B 0,C 180,E1 3499.697,E2 3499.697} C_VEL
LIN {X 0,Y 698.871,Z 1226.068,A -85,B 0,C 180,E1 3503.151,E2 3503.151} C_VEL
LIN {X 0,Y 698.77,Z 1232.652,A -85,B 0,C 180,E1 3506.27,E2 3506.27} C_VEL
LIN {X 0,Y 698.805,Z 1235.5,A -85,B 0,C 180,E1 3510,E2 3510} C_VEL
LIN {X 0,Y 698.801,Z 1232.652,A -85,B 0,C 180,E1 3513.73,E2 3513.73} C_VEL
LIN {X 0,Y 698.847,Z 1226.069,A -85,B 0,C 180,E1 3516.849,E2 3516.849} C_VEL
LIN {X 0,Y 698.981,Z 1213.837,A -85,B 0,C 180,E1 3520.303,E2 3520.303} C_VEL
LIN {X 0,Y 699.231,Z 1197.74,A -85,B 0,C 180,E1 3523.524,E2 3523.524} C_VEL
LIN {X 0,Y 699.741,Z 1175.55,A -85,B 0,C 180,E1 3526.836,E2 3526.836} C_VEL
LIN {X 0,Y 700.611,Z 1149.539,A -85,B 0,C 180,E1 3529.868,E2 3529.868} C_VEL
LIN {X 0,Y 701.853,Z 1116.881,A -85,B 0,C 180,E1 3532.868,E2 3532.868} C_VEL
LIN {X 0,Y 703.387,Z 1078.751,A -85,B 0,C 180,E1 3535.597,E2 3535.597} C_VEL
LIN {X 0,Y 704.976,Z 1037.162,A -85,B 0,C 180,E1 3537.872,E2 3537.872} C_VEL
LIN {X 0,Y 706.377,Z 995.216,A -85,B 0,C 180,E1 3539.563,E2 3539.563} C_VEL
LIN {X 0,Y 707.457,Z 954.996,A -85,B 0,C 180,E1 3540.711,E2 3540.711} C_VEL
LIN {X 0,Y 708.114,Z 911.667,A -85,B 0,C 180,E1 3541.471,E2 3541.471} C_VEL
LIN {X 0,Y 707.532,Z 879.91,A -85,B 0,C 180,E1 3541.879,E2 3541.879} C_VEL
LIN {X 0,Y 698.497,Z 859.31,A -85,B 0,C 180,E1 3542.63,E2 3542.63} C_VEL
LIN {X 0,Y 698.378,Z 859.31,A -85,B 0,C 180,E1 3547.411,E2 3547.411} C_VEL
LIN {X 0,Y 698.381,Z 859.31,A -85,B 0,C 180,E1 3552.478,E2 3552.478} C_VEL
LIN {X 0,Y 698.219,Z 859.31,A -85,B 0,C 180,E1 3557.73,E2 3557.73} C_VEL
LIN {X 0,Y 698.227,Z 859.31,A -85,B 0,C 180,E1 3562.589,E2 3562.589} C_VEL
LIN {X 0,Y 698.313,Z 859.31,A -85,B 0,C 180,E1 3567.808,E2 3567.808} C_VEL
LIN {X 0,Y 698.435,Z 859.31,A -85,B 0,C 180,E1 3572.902,E2 3572.902} C_VEL
LIN {X 0,Y 698.536,Z 859.31,A -85,B 0,C 180,E1 3577.021,E2 3577.021} C_VEL
LIN {X 0,Y 698.549,Z 859.31,A -85,B 0,C 180,E1 3582.639,E2 3582.639} C_VEL
LIN {X 0,Y 698.38,Z 859.31,A -85,B 0,C 180,E1 3587.52,E2 3587.52} C_VEL
LIN {X 0,Y 698.626,Z 859.31,A -85,B 0,C 180,E1 3592.523,E2 3592.523} C_VEL
LIN {X 0,Y 698.756,Z 859.31,A -85,B 0,C 180,E1 3597.513,E2 3597.513} C_VEL
LIN {X 0,Y 698.626,Z 859.31,A -85,B 0,C 180,E1 3602.484,E2 3602.484} C_VEL
LIN {X 0,Y 698.585,Z 859.31,A -85,B 0,C 180,E1 3606.223,E2 3606.223} C_VEL
LIN {X 0,Y 698.5,Z 859.31,A -85,B 0,C 180,E1 3611.254,E2 3611.254} C_VEL
LIN {X 0,Y 698.545,Z 859.31,A -85,B 0,C 180,E1 3616.373,E2 3616.373} C_VEL
LIN {X 0,Y 698.44,Z 859.31,A -85,B 0,C 180,E1 3621.635,E2 3621.635} C_VEL
LIN {X 0,Y 698.409,Z 859.31,A -85,B 0,C 180,E1 3625.708,E2 3625.708} C_VEL
LIN {X 0,Y 698.321,Z 859.31,A -85,B 0,C 180,E1 3629.928,E2 3629.928} C_VEL
LIN {X 0,Y 698.278,Z 859.31,A -85,B 0,C 180,E1 3634.451,E2 3634.451} C_VEL
LIN {X 0,Y 698.239,Z 859.31,A -85,B 0,C 180,E1 3638.987,E2 3638.987} C_VEL
LIN {X 0,Y 698.166,Z 859.31,A -85,B 0,C 180,E1 3644.256,E2 3644.256} C_VEL
LIN {X 0,Y 698.213,Z 859.31,A -85,B 0,C 180,E1 3649.407,E2 3649.407} C_VEL
LIN {X 0,Y 698.395,Z 859.31,A -85,B 0,C 180,E1 3654.14,E2 3654.14} C_VEL
LIN {X 0,Y 698.259,Z 859.31,A -85,B 0,C 180,E1 3658.613,E2 3658.613} C_VEL
LIN {X 0,Y 698.417,Z 859.31,A -85,B 0,C 180,E1 3664.055,E2 3664.055} C_VEL
LIN {X 0,Y 704.952,Z 877.807,A -85,B 0,C 180,E1 3664.539,E2 3664.539} C_VEL
LIN {X 0,Y 704.524,Z 968.016,A -85,B 0,C 180,E1 3665.602,E2 3665.602} C_VEL
LIN {X 0,Y 703.828,Z 1007.584,A -85,B 0,C 180,E1 3666.55,E2 3666.55} C_VEL
LIN {X 0,Y 702.849,Z 1044.875,A -85,B 0,C 180,E1 3667.937,E2 3667.937} C_VEL
LIN {X 0,Y 701.751,Z 1081.444,A -85,B 0,C 180,E1 3669.853,E2 3669.853} C_VEL
LIN {X 0,Y 700.709,Z 1113.865,A -85,B 0,C 180,E1 3672.147,E2 3672.147} C_VEL
LIN {X 0,Y 699.919,Z 1142.139,A -85,B 0,C 180,E1 3674.79,E2 3674.79} C_VEL
LIN {X 0,Y 699.375,Z 1165.217,A -85,B 0,C 180,E1 3677.646,E2 3677.646} C_VEL
LIN {X 0,Y 699.058,Z 1182.602,A -85,B 0,C 180,E1 3680.56,E2 3680.56} C_VEL
LIN {X 0,Y 698.907,Z 1194.777,A -85,B 0,C 180,E1 3683.464,E2 3683.464} C_VEL
LIN {X 0,Y 698.874,Z 1202.017,A -85,B 0,C 180,E1 3686.271,E2 3686.271} C_VEL
LIN {X 0,Y 698.805,Z 1205.12,A -85,B 0,C 180,E1 3688.758,E2 3688.758} C_VEL
LIN {X 0,Y 698.89,Z 1205.045,A -85,B 0,C 180,E1 3691.243,E2 3691.243} C_VEL
LIN {X 0,Y 698.93,Z 1200.385,A -85,B 0,C 180,E1 3694.444,E2 3694.444} C_VEL
LIN {X 0,Y 699.074,Z 1189.734,A -85,B 0,C 180,E1 3697.786,E2 3697.786} C_VEL
LIN {X 0,Y 699.257,Z 1173.877,A -85,B 0,C 180,E1 3700.93,E2 3700.93} C_VEL
LIN {X 0,Y 699.685,Z 1152.473,A -85,B 0,C 180,E1 3703.942,E2 3703.942} C_VEL
LIN {X 0,Y 700.37,Z 1126.6,A -85,B 0,C 180,E1 3706.659,E2 3706.659} C_VEL
LIN {X 0,Y 701.302,Z 1096.615,A -85,B 0,C 180,E1 3709.058,E2 3709.058} C_VEL
LIN {X 0,Y 702.302,Z 1062.879,A -85,B 0,C 180,E1 3711.104,E2 3711.104} C_VEL
LIN {X 0,Y 703.313,Z 1025.506,A -85,B 0,C 180,E1 3712.76,E2 3712.76} C_VEL
LIN {X 0,Y 704.245,Z 985.298,A -85,B 0,C 180,E1 3713.961,E2 3713.961} C_VEL
LIN {X 0,Y 704.666,Z 943.371,A -85,B 0,C 180,E1 3714.659,E2 3714.659} C_VEL
LIN {X 0,Y 704.377,Z 876.243,A -85,B 0,C 180,E1 3715.411,E2 3715.411} C_VEL
LIN {X 0,Y 698.326,Z 859.31,A -85,B 0,C 180,E1 3715.893,E2 3715.893} C_VEL
LIN {X 0,Y 698.33,Z 859.31,A -85,B 0,C 180,E1 3719.939,E2 3719.939} C_VEL
LIN {X 0,Y 698.325,Z 859.31,A -85,B 0,C 180,E1 3724.481,E2 3724.481} C_VEL
LIN {X 0,Y 698.273,Z 859.31,A -85,B 0,C 180,E1 3729,E2 3729} C_VEL
LIN {X 0,Y 698.143,Z 859.31,A -85,B 0,C 180,E1 3734.272,E2 3734.272} C_VEL
LIN {X 0,Y 698.171,Z 859.31,A -85,B 0,C 180,E1 3739.432,E2 3739.432} C_VEL
LIN {X 0,Y 698.399,Z 859.31,A -85,B 0,C 180,E1 3744.153,E2 3744.153} C_VEL
LIN {X 0,Y 698.23,Z 859.31,A -85,B 0,C 180,E1 3748.622,E2 3748.622} C_VEL
LIN {X 0,Y 698.373,Z 859.31,A -85,B 0,C 180,E1 3752.903,E2 3752.903} C_VEL
LIN {X 0,Y 698.465,Z 859.31,A -85,B 0,C 180,E1 3757.023,E2 3757.023} C_VEL
LIN {X 0,Y 698.307,Z 859.31,A -85,B 0,C 180,E1 3761.012,E2 3761.012} C_VEL
LIN {X 0,Y 698.372,Z 859.31,A -85,B 0,C 180,E1 3766.197,E2 3766.197} C_VEL
LIN {X 0,Y 698.578,Z 859.31,A -85,B 0,C 180,E1 3771.271,E2 3771.271} C_VEL
LIN {X 0,Y 698.714,Z 859.31,A -85,B 0,C 180,E1 3776.272,E2 3776.272} C_VEL
LIN {X 0,Y 698.86,Z 859.31,A -85,B 0,C 180,E1 3781.244,E2 3781.244} C_VEL
LIN {X 0,Y 698.588,Z 859.31,A -85,B 0,C 180,E1 3786.226,E2 3786.226} C_VEL
LIN {X 0,Y 698.478,Z 859.31,A -85,B 0,C 180,E1 3791.258,E2 3791.258} C_VEL
LIN {X 0,Y 698.514,Z 859.31,A -85,B 0,C 180,E1 3796.076,E2 3796.076} C_VEL
LIN {X 0,Y 696.03,Z 859.31,A -85,B 0,C 180,E1 3797.136,E2 3797.136} C_VEL
LIN {X 0,Y 690.664,Z 859.31,A -85,B 0,C 180,E1 3798.719,E2 3798.719} C_VEL
LIN {X 0,Y 690.58,Z 859.31,A -85,B 0,C 180,E1 3798.902,E2 3798.902} C_VEL
LIN {X 0,Y 690.553,Z 859.31,A -85,B 0,C 180,E1 3803.26,E2 3803.26} C_VEL
LIN {X 0,Y 690.499,Z 859.31,A -85,B 0,C 180,E1 3808.622,E2 3808.622} C_VEL
LIN {X 0,Y 690.36,Z 859.31,A -85,B 0,C 180,E1 3813.48,E2 3813.48} C_VEL
LIN {X 0,Y 690.395,Z 859.31,A -85,B 0,C 180,E1 3817.909,E2 3817.909} C_VEL
LIN {X 0,Y 690.252,Z 859.31,A -85,B 0,C 180,E1 3823.577,E2 3823.577} C_VEL
LIN {X 0,Y 690.209,Z 859.31,A -85,B 0,C 180,E1 3828.805,E2 3828.805} C_VEL
LIN {X 0,Y 690.528,Z 859.31,A -85,B 0,C 180,E1 3834.266,E2 3834.266} C_VEL
LIN {X 0,Y 690.576,Z 859.711,A -85,B 0,C 180,E1 3836.997,E2 3836.997} C_VEL
LIN {X 0,Y 701.539,Z 885.06,A -85,B 0,C 180,E1 3837.877,E2 3837.877} C_VEL
LIN {X 0,Y 700.939,Z 941.38,A -85,B 0,C 180,E1 3838.661,E2 3838.661} C_VEL
LIN {X 0,Y 699.544,Z 986.34,A -85,B 0,C 180,E1 3839.81,E2 3839.81} C_VEL
LIN {X 0,Y 698.146,Z 1028.54,A -85,B 0,C 180,E1 3841.426,E2 3841.426} C_VEL
LIN {X 0,Y 696.444,Z 1068.896,A -85,B 0,C 180,E1 3843.511,E2 3843.511} C_VEL
LIN {X 0,Y 694.784,Z 1107.518,A -85,B 0,C 180,E1 3846.126,E2 3846.126} C_VEL
LIN {X 0,Y 693.338,Z 1142.637,A -85,B 0,C 180,E1 3849.198,E2 3849.198} C_VEL
LIN {X 0,Y 692.166,Z 1171.875,A -85,B 0,C 180,E1 3852.481,E2 3852.481} C_VEL
LIN {X 0,Y 691.453,Z 1196.133,A -85,B 0,C 180,E1 3856.051,E2 3856.051} C_VEL
LIN {X 0,Y 691.143,Z 1213.835,A -85,B 0,C 180,E1 3859.579,E2 3859.579} C_VEL
LIN {X 0,Y 690.996,Z 1226.068,A -85,B 0,C 180,E1 3863.073,E2 3863.073} C_VEL
LIN {X 0,Y 690.888,Z 1232.651,A -85,B 0,C 180,E1 3866.227,E2 3866.227} C_VEL
LIN {X 0,Y 690.908,Z 1235.5,A -85,B 0,C 180,E1 3870,E2 3870} C_VEL
LIN {X 0,Y 690.916,Z 1232.652,A -85,B 0,C 180,E1 3873.772,E2 3873.772} C_VEL
LIN {X 0,Y 690.966,Z 1226.069,A -85,B 0,C 180,E1 3876.927,E2 3876.927} C_VEL
LIN {X 0,Y 691.121,Z 1213.838,A -85,B 0,C 180,E1 3880.421,E2 3880.421} C_VEL
LIN {X 0,Y 691.4,Z 1197.569,A -85,B 0,C 180,E1 3883.711,E2 3883.711} C_VEL
LIN {X 0,Y 692.033,Z 1174.336,A -85,B 0,C 180,E1 3887.193,E2 3887.193} C_VEL
LIN {X 0,Y 693.03,Z 1147.509,A -85,B 0,C 180,E1 3890.306,E2 3890.306} C_VEL
LIN {X 0,Y 694.378,Z 1115.66,A -85,B 0,C 180,E1 3893.228,E2 3893.228} C_VEL
LIN {X 0,Y 696.061,Z 1078.81,A -85,B 0,C 180,E1 3895.882,E2 3895.882} C_VEL
LIN {X 0,Y 697.825,Z 1037.533,A -85,B 0,C 180,E1 3898.164,E2 3898.164} C_VEL
LIN {X 0,Y 699.435,Z 995.213,A -85,B 0,C 180,E1 3899.886,E2 3899.886} C_VEL
LIN {X 0,Y 700.63,Z 955.458,A -85,B 0,C 180,E1 3901.032,E2 3901.032} C_VEL
LIN {X 0,Y 701.411,Z 910.746,A -85,B 0,C 180,E1 3901.82,E2 3901.82} C_VEL
LIN {X 0,Y 700.897,Z 882.611,A -85,B 0,C 180,E1 3902.185,E2 3902.185} C_VEL
LIN {X 0,Y 690.535,Z 859.31,A -85,B 0,C 180,E1 3903.046,E2 3903.046} C_VEL
LIN {X 0,Y 690.41,Z 859.31,A -85,B 0,C 180,E1 3907.918,E2 3907.918} C_VEL
LIN {X 0,Y 690.488,Z 859.31,A -85,B 0,C 180,E1 3913.612,E2 3913.612} C_VEL
LIN {X 0,Y 690.268,Z 859.31,A -85,B 0,C 180,E1 3918.82,E2 3918.82} C_VEL
LIN {X 0,Y 690.316,Z 859.31,A -85,B 0,C 180,E1 3924.309,E2 3924.309} C_VEL
LIN {X 0,Y 690.405,Z 859.31,A -85,B 0,C 180,E1 3929.689,E2 3929.689} C_VEL
LIN {X 0,Y 690.6,Z 859.31,A -85,B 0,C 180,E1 3934.106,E2 3934.106} C_VEL
LIN {X 0,Y 690.562,Z 859.31,A -85,B 0,C 180,E1 3939.45,E2 3939.45} C_VEL
LIN {X 0,Y 690.577,Z 859.31,A -85,B 0,C 180,E1 3944.736,E2 3944.736} C_VEL
LIN {X 0,Y 690.701,Z 859.31,A -85,B 0,C 180,E1 3949.893,E2 3949.893} C_VEL
LIN {X 0,Y 690.704,Z 859.31,A -85,B 0,C 180,E1 3954.965,E2 3954.965} C_VEL
LIN {X 0,Y 690.796,Z 859.31,A -85,B 0,C 180,E1 3959.998,E2 3959.998} C_VEL
LIN {X 0,Y 690.922,Z 859.31,A -85,B 0,C 180,E1 3965.03,E2 3965.03} C_VEL
LIN {X 0,Y 690.628,Z 859.31,A -85,B 0,C 180,E1 3970.105,E2 3970.105} C_VEL
LIN {X 0,Y 690.602,Z 859.31,A -85,B 0,C 180,E1 3975.26,E2 3975.26} C_VEL
LIN {X 0,Y 690.586,Z 859.31,A -85,B 0,C 180,E1 3980.545,E2 3980.545} C_VEL
LIN {X 0,Y 690.482,Z 859.31,A -85,B 0,C 180,E1 3986.025,E2 3986.025} C_VEL
LIN {X 0,Y 690.403,Z 859.31,A -85,B 0,C 180,E1 3991.133,E2 3991.133} C_VEL
LIN {X 0,Y 690.407,Z 859.31,A -85,B 0,C 180,E1 3996.328,E2 3996.328} C_VEL
LIN {X 0,Y 690.261,Z 859.31,A -85,B 0,C 180,E1 4001.722,E2 4001.722} C_VEL
LIN {X 0,Y 690.262,Z 859.31,A -85,B 0,C 180,E1 4007.116,E2 4007.116} C_VEL
LIN {X 0,Y 690.432,Z 859.31,A -85,B 0,C 180,E1 4012.172,E2 4012.172} C_VEL
LIN {X 0,Y 690.382,Z 859.31,A -85,B 0,C 180,E1 4016.721,E2 4016.721} C_VEL
LIN {X 0,Y 690.412,Z 859.31,A -85,B 0,C 180,E1 4021.359,E2 4021.359} C_VEL
LIN {X 0,Y 690.509,Z 859.31,A -85,B 0,C 180,E1 4023.746,E2 4023.746} C_VEL
LIN {X 0,Y 697.826,Z 881.344,A -85,B 0,C 180,E1 4024.3,E2 4024.3} C_VEL
LIN {X 0,Y 697.317,Z 969.456,A -85,B 0,C 180,E1 4025.359,E2 4025.359} C_VEL
LIN {X 0,Y 696.479,Z 1009.885,A -85,B 0,C 180,E1 4026.358,E2 4026.358} C_VEL
LIN {X 0,Y 695.265,Z 1049.515,A -85,B 0,C 180,E1 4027.902,E2 4027.902} C_VEL
LIN {X 0,Y 694.113,Z 1084.634,A -85,B 0,C 180,E1 4029.83,E2 4029.83} C_VEL
LIN {X 0,Y 692.94,Z 1116.587,A -85,B 0,C 180,E1 4032.173,E2 4032.173} C_VEL
LIN {X 0,Y 692.103,Z 1143.526,A -85,B 0,C 180,E1 4034.768,E2 4034.768} C_VEL
LIN {X 0,Y 691.526,Z 1166.304,A -85,B 0,C 180,E1 4037.664,E2 4037.664} C_VEL
LIN {X 0,Y 691.164,Z 1184.422,A -85,B 0,C 180,E1 4040.829,E2 4040.829} C_VEL
LIN {X 0,Y 690.995,Z 1195.74,A -85,B 0,C 180,E1 4043.705,E2 4043.705} C_VEL
LIN {X 0,Y 690.985,Z 1202.017,A -85,B 0,C 180,E1 4046.228,E2 4046.228} C_VEL
LIN {X 0,Y 690.912,Z 1205.12,A -85,B 0,C 180,E1 4048.743,E2 4048.743} C_VEL
LIN {X 0,Y 690.992,Z 1205.046,A -85,B 0,C 180,E1 4051.257,E2 4051.257} C_VEL
LIN {X 0,Y 691.031,Z 1200.387,A -85,B 0,C 180,E1 4054.495,E2 4054.495} C_VEL
LIN {X 0,Y 691.168,Z 1189.736,A -85,B 0,C 180,E1 4057.876,E2 4057.876} C_VEL
LIN {X 0,Y 691.433,Z 1173.88,A -85,B 0,C 180,E1 4061.056,E2 4061.056} C_VEL
LIN {X 0,Y 691.878,Z 1152.476,A -85,B 0,C 180,E1 4064.102,E2 4064.102} C_VEL
LIN {X 0,Y 692.662,Z 1126.605,A -85,B 0,C 180,E1 4066.85,E2 4066.85} C_VEL
LIN {X 0,Y 693.677,Z 1096.758,A -85,B 0,C 180,E1 4069.266,E2 4069.266} C_VEL
LIN {X 0,Y 694.848,Z 1062.885,A -85,B 0,C 180,E1 4071.341,E2 4071.341} C_VEL
LIN {X 0,Y 695.936,Z 1026.462,A -85,B 0,C 180,E1 4072.978,E2 4072.978} C_VEL
LIN {X 0,Y 696.979,Z 987.393,A -85,B 0,C 180,E1 4074.173,E2 4074.173} C_VEL
LIN {X 0,Y 697.52,Z 945.473,A -85,B 0,C 180,E1 4074.906,E2 4074.906} C_VEL
